// TwinCAT 3 PLC project Resi4MPM_Lib
// Title: Resi4MPM
// Company: Jan Wilch
// ProjectVersion: 1.0.0
// ProgramVersion: 3.1.4026.11
// libraries:
//   Tc2_Standard, * (Beckhoff Automation GmbH)
//   Tc2_System, * (Beckhoff Automation GmbH)
//   Tc3_Module, * (Beckhoff Automation GmbH)
// project tree:
//   Models/Behavior/ BehaviorBase.TcPOU, ControlPrimitiveBase.TcPOU, EBehaviorType.TcDUT, EOperationResult.TcDUT, ESpecialBehaviorIds.TcDUT, LinearSequence.TcPOU, ModuleSequenceBase.TcPOU
//   Models/Behavior/Strategy/ ESpecialStepIds.TcDUT, EStrategyStates.TcDUT, SStep.TcDUT, SStrategy.TcDUT, STransition.TcDUT
//   Models/ProcessState/AdsStateSynch/ SAdsSymbol.TcDUT
//   Models/ProcessState/ EDataType.TcDUT, HardwareObservationBase.TcPOU, ParameterSet.TcPOU, ProcessState.TcPOU, ProductBase.TcPOU, SNamedValue.TcDUT, SValue.TcDUT, UValues.TcDUT
//   Models/ProcessState/ProcessCondition/ BoolExpression.TcPOU, ComparisonExpression.TcPOU, EBoolOperation.TcDUT, EComparisonType.TcDUT, EExpressionType.TcDUT, IExpression.TcIO, IValExp.TcIO, SPrimitiveCondition.TcDUT, SBoolExpressionSpec.TcDUT, SInterlock.TcDUT, SConditionSpec.TcDUT, ValueExpression.TcPOU
//   Models/Reconfiguration/ EAbortState.TcDUT, ECompSeqState.TcDUT, ERecoveryState.TcDUT, ERetargetType.TcDUT, SCompensation.TcDUT, SRecovery.TcDUT, SRecoveryRequestOutput.TcDUT, SRetargeting.TcDUT, STriggeredOutput.TcDUT
//   / ResiConst.TcGVL
//   Services/Base/ ErrorManagerBase.TcPOU, ESeverity.TcDUT, ESpecialAlarmIds.TcDUT, IService.TcIO, SAlarm.TcDUT
//   Services/ ProcessManager.TcPOU, ServiceContainer.TcPOU, StateTracker.TcPOU
// real-time tasks:
//   TASK PlcTask: cycle T#10ms, priority 20, ADS port 350
//   TASK PlcTask1: cycle T#10ms, priority 23, ADS port 351
//   TASK PlcTask2: cycle T#10ms, priority 22, ADS port 352
//   TASK PlcTask3: cycle T#10ms, priority 21, ADS port 353

// ---- Models/Behavior/EBehaviorType.TcDUT
{attribute 'qualified_only'}
{attribute 'strict'}
TYPE EBehaviorType :
(
	none := 0,
	control_primitive := 1,
	user_sequence := 2,
	generated_sequence := 3
);
END_TYPE

// ---- Models/Behavior/EOperationResult.TcDUT
{attribute 'qualified_only'}
{attribute 'strict'}
TYPE EOperationResult :
(
	none := 0,
	success := 1,
	busy := 2,
	recovering := 3,
	waiting := 4,
	failed := 5,
	synced_success := 6
);
END_TYPE

// ---- Models/Behavior/ESpecialBehaviorIds.TcDUT
{attribute 'qualified_only'}
{attribute 'strict'}
TYPE ESpecialBehaviorIds :
(
	empty := 0,
	max_id := ResiConst.BEHAVIORS_ARR_MAX
) UINT;
END_TYPE

// ---- Models/Behavior/Strategy/ESpecialStepIds.TcDUT
{attribute 'qualified_only'}
{attribute 'strict'}
TYPE ESpecialStepIds :
(
	unset := -1,
	start := 0,
	end := 1
) INT;
END_TYPE

// ---- Models/Behavior/Strategy/EStrategyStates.TcDUT
{attribute 'qualified_only'}
{attribute 'strict'}
{attribute 'to_string'}
TYPE EStrategyStates :
(
	none := 0,
	ready := 1,
	running := 2,
	halting := 3,
	halted := 4,
	done := 5
) USINT;
END_TYPE

// ---- Models/Behavior/Strategy/SStep.TcDUT
{attribute 'OPC.UA.DA.StructuredType' := '1'}
TYPE SStep :
STRUCT
	// Set by the RA
	BehaviorType: EBehaviorType;
	BehaviorId: UINT;
	Parameters: ParameterSet;
	
	// defines ADS connections to step states on partner PLCs
	ExtSymbols: ARRAY [ResiConst.ARR_MIN..ResiConst.MAX_SYNC_PARTNERS] OF SAdsSymbol;
	// index of the responsible PLC (-1 is the current PLC is responsible)
	ExecutorIdx: INT;
	
	// Set by the PLC, read-only
	{attribute 'OPC.UA.DA.Access' := '1'}
	State: EOperationResult;
END_STRUCT
END_TYPE

// ---- Models/Behavior/Strategy/SStrategy.TcDUT
TYPE SStrategy :
STRUCT
	State: EStrategyStates;
	
	LoopStrategy: BOOL;
	Steps: ARRAY [ResiConst.ARR_MIN..ResiConst.STRAT_LEN_MAX] OF SStep;
	Transitions: ARRAY [ResiConst.ARR_MIN..ResiConst.STRAT_LEN_MAX] OF STransition;
	
	IsMaster: BOOL;
	NumPartners: UINT;
END_STRUCT
END_TYPE

// ---- Models/Behavior/Strategy/STransition.TcDUT
{attribute 'OPC.UA.DA.StructuredType' := '1'}
TYPE STransition :
STRUCT
	// determines whether this transition in a SStrategy's transition array is part of the strategy.
	IsSet: BOOL;
	
	// -1 signifies unset (because ID 0 is the start node)
	PrevStepIds: ARRAY [ResiConst.ARR_MIN..ResiConst.STRAT_PARALLEL_MAX] OF INT;
	// -1 signifies unset (because ID 0 is the start node)	
	NextStepIds: ARRAY [ResiConst.ARR_MIN..ResiConst.STRAT_PARALLEL_MAX] OF INT;
	
	ExpressionType: EExpressionType;
	ExpressionIdx: UINT;
END_STRUCT
END_TYPE

// ---- Models/ProcessState/AdsStateSynch/SAdsSymbol.TcDUT
TYPE SAdsSymbol :
STRUCT
	IsSet: BOOL;		// indicates whether this target is defined
	DataType: EDataType;
	
	NetId: T_AmsNetID;	// alias for STRING(23)
	Port: T_AmsPort;	// alias for UINT
	
	IdxGrp: UDINT;
	IdxOffs: UDINT;
END_STRUCT
END_TYPE

// ---- Models/ProcessState/EDataType.TcDUT
{attribute 'qualified_only'}
TYPE EDataType :
(
	none := 0,
	dont_care := 1,
	binary := 2,
	numeric := 3,
	string_t := 4
) USINT;
END_TYPE

// ---- Models/ProcessState/ProcessCondition/EBoolOperation.TcDUT
{attribute 'qualified_only'}
{attribute 'strict'}
TYPE EBoolOperation :
(
	none := 0,
	and_op := 1,
	nand_op := 2,
	or_op := 3,
	nor_op := 4
);
END_TYPE

// ---- Models/ProcessState/ProcessCondition/EComparisonType.TcDUT
{attribute 'qualified_only'}
{attribute 'strict'}
TYPE EComparisonType :
(
	none := 0,
	equals := 1,
	not_equal := 2,
	greater := 3,
	less := 4,
	greater_eq := 5,
	less_eq := 6
);
END_TYPE

// ---- Models/ProcessState/ProcessCondition/EExpressionType.TcDUT
{attribute 'qualified_only'}
{attribute 'strict'}
TYPE EExpressionType :
(
	none := 0,
	boolean := 1,
	comparison := 2,
	value := 3
);
END_TYPE

// ---- Models/ProcessState/ProcessCondition/SPrimitiveCondition.TcDUT
TYPE SPrimitiveCondition EXTENDS SConditionSpec :
STRUCT
	PrimitiveId: UINT;
	// if it's not a precondition, it's a postcondition
	IsPre: BOOL;
END_STRUCT
END_TYPE

// ---- Models/ProcessState/ProcessCondition/SBoolExpressionSpec.TcDUT
{attribute 'OPC.UA.DA.StructuredType' := '1'}
TYPE SBoolExpressionSpec :
STRUCT
	Operator: EBoolOperation;
	
	LeftType: EExpressionType;
	LeftIdx: UINT;
	
	RightType: EExpressionType;
	RightIdx: UINT;
END_STRUCT
END_TYPE

// ---- Models/ProcessState/ProcessCondition/SInterlock.TcDUT
TYPE SInterlock EXTENDS SConditionSpec :
STRUCT
	DefaultValue: BOOL;
END_STRUCT
END_TYPE

// ---- Models/ProcessState/ProcessCondition/SConditionSpec.TcDUT
{attribute 'OPC.UA.DA.StructuredType' := '1'}
TYPE SConditionSpec :
STRUCT
	IsActive: BOOL;
	ExpressionType: EExpressionType;
	ExpressionIdx: UINT;
END_STRUCT
END_TYPE

// ---- Models/ProcessState/SNamedValue.TcDUT
{attribute 'OPC.UA.DA.StructuredType' := '1'}
TYPE SNamedValue EXTENDS SValue :
STRUCT
	Name: STRING;
END_STRUCT
END_TYPE

// ---- Models/ProcessState/SValue.TcDUT
TYPE SValue :
STRUCT
	DataType: EDataType;
	Value: UValues;
	Defined: BOOL;
END_STRUCT
END_TYPE

// ---- Models/ProcessState/UValues.TcDUT
TYPE UValues :
UNION
	Binary: BOOL;
	Numeric: LREAL;
	String_t: STRING;
END_UNION
END_TYPE

// ---- Models/Reconfiguration/EAbortState.TcDUT
{attribute 'qualified_only'}
{attribute 'strict'}
TYPE EAbortState :
(
	none := 0,
	requested := 1,
	aborting := 2,
	aborted := 3
);
END_TYPE

// ---- Models/Reconfiguration/ECompSeqState.TcDUT
{attribute 'qualified_only'}
{attribute 'strict'}
TYPE ECompSeqState :
(
	none := 0,
	preparing := 1,
	running := 2,
	finished := 3
);
END_TYPE

// ---- Models/Reconfiguration/ERecoveryState.TcDUT
{attribute 'qualified_only'}
{attribute 'strict'}
TYPE ERecoveryState :
(
	none := 0,
	requested := 1,
	awaiting := 2,
	running := 3,
	completed := 4,
	failed := 5
);
END_TYPE

// ---- Models/Reconfiguration/ERetargetType.TcDUT
{attribute 'qualified_only'}
{attribute 'strict'}
TYPE ERetargetType :
(
	not_retargeted := 0,
	primitive_target := 1,
	sequence_target := 2
);
END_TYPE

// ---- Models/Reconfiguration/SCompensation.TcDUT
{attribute 'OPC.UA.DA.StructuredType' := '1'}
TYPE SCompensation :
STRUCT
	IsActive: BOOL;	

	(* ID of the Control Primitive that cannot operate anymore. *)
	SickPrimitiveId: UINT;
	
	(* Specifies whether the sick primitive is replaced by another primitive or a sequence. *)
	NewType: EBehaviorType;
	
	(* If NewType is primitive or user-sequence: ID of the sick primitive's replacement. *)
	NewId: UINT;
	
	(* If needed, parameters that are set (or overwritten) before executing the replacement.
	   For replacement types primtive or user-generated sequence, only the first element is used. *)
	ParameterSets: ARRAY [ResiConst.ARR_MIN..ResiConst.MODULE_SEQ_ARR_MAX] OF ParameterSet;
	
	(* If NewType is generated sequence: The (linear) sequence of copmensation primitives. *)
	PrimitiveIds: ARRAY [ResiConst.ARR_MIN..ResiConst.MODULE_SEQ_ARR_MAX] OF UINT;
END_STRUCT
END_TYPE

// ---- Models/Reconfiguration/SRecovery.TcDUT
{attribute 'OPC.UA.DA.StructuredType' := '1'}
TYPE SRecovery :
STRUCT
	(* The sequence of Control Primitives to execute for recovery or defining.*)
	RecoveryStrategy: ARRAY [ResiConst.ARR_MIN..ResiConst.MODULE_SEQ_ARR_MAX] OF UINT;
	
	(* The parameters needed by the strategy's primitives. *)
	RecoveryParameters: ParameterSet;
END_STRUCT
END_TYPE

// ---- Models/Reconfiguration/SRecoveryRequestOutput.TcDUT
{attribute 'OPC.UA.DA.StructuredType' := '1'}
TYPE SRecoveryRequestOutput EXTENDS STriggeredOutput :
STRUCT
	RequestedState: STRING(256);
END_STRUCT
END_TYPE

// ---- Models/Reconfiguration/SRetargeting.TcDUT
TYPE SRetargeting :
STRUCT
	RetargetType: ERetargetType;
	TargetId: UINT;
	// parameters that are set or overwritten before the primitive is executed
	OverwriteParams: ParameterSet;
END_STRUCT
END_TYPE

// ---- Models/Reconfiguration/STriggeredOutput.TcDUT
TYPE STriggeredOutput :
STRUCT
	ChangeTrigger: USINT;
END_STRUCT
END_TYPE

// ---- Services/Base/ESeverity.TcDUT
{attribute 'qualified_only'}
{attribute 'strict'}
TYPE ESeverity :
(
	none := 0,
	info := 1,
	warning := 2,
	error := 3
) UINT;
END_TYPE

// ---- Services/Base/ESpecialAlarmIds.TcDUT
{attribute 'qualified_only'}
{attribute 'strict'}
TYPE ESpecialAlarmIds :
(
	none := 0,
	recovery_request := 990,
	definition_request := 991,
	strategy_received := 992
) UINT;
END_TYPE

// ---- Services/Base/SAlarm.TcDUT
(*
 * see: https://www.plcnext.help/te/Service_Components/Alarms/Alarms_via_OPC_UA.htm
 *)
{attribute 'OPC.UA.DA.StructuredType' := '1'}
TYPE SAlarm :
STRUCT
	// Time in number of 100 ns intervals since 01.01.1601.
	TimeTicks: ULINT;
	AlarmId: UINT;
	// TODO - AlarmType
	Active: BOOL;
	//Acknowledged: BOOL;
	//Confirmed: BOOL;
	Severity: ESeverity;
	//RetainAlarm: BOOL;
	Message: STRING;
	InstanceName: STRING;
END_STRUCT
END_TYPE

// ---- ResiConst.TcGVL
{attribute 'qualified_only'}
VAR_GLOBAL CONSTANT	
	// Lower bound of all Resi4MPM arrays.
	ARR_MIN: UINT := 0;
	// Default upper bound of Resi4MPM arrays.
	DEFAULT_ARR_MAX: UINT := 10;
	// Max length of behaviors (separately length of Control Primitives and Module Sequences).
	BEHAVIORS_ARR_MAX: UINT := 100;
	// Max length of observed process variables.
	STATE_ARR_MAX: UINT := 150;
	// Max length of units observing the process state.
	OBSERVERS_ARR_MAX: UINT := 100;
	// Max length of UC-C strategies introduced at runtime.
	COMPENSATIONS_ARR_MAX: UINT := 10;
	// Max Control Primitive count of Module Sequences.
	MODULE_SEQ_ARR_MAX: UINT := 10;
	// Max number of parameters for a Behavior.
	PARAMS_ARR_MAX: UINT := 10;
	// Max number of Products 
	PRODUCTS_ARR_MAX: UINT := 20;
	// Max number of parallel steps in a runtime-defined strategy.
	STRAT_PARALLEL_MAX: UINT := 5;
	// Max length (number of steps/transitions) of a runtime-defined strategy.
	STRAT_LEN_MAX: UINT := 24;
	// Max length of runtime-changeable expressions.
	RT_EXPRS_MAX: UINT := 24;
	// Maximum number of synchronized foreign PLCs.
	MAX_SYNC_PARTNERS: UINT := 5;
END_VAR

// ---- Models/ProcessState/ProcessCondition/IExpression.TcIO
INTERFACE IExpression EXTENDS __System.IQueryInterface

METHOD IsTrue : BOOL
VAR_INPUT
	i_ptrProcessState: POINTER TO ProcessState;
END_VAR
END_METHOD

METHOD ToString : STRING(256)
VAR_INPUT
END_VAR
END_METHOD

END_INTERFACE

// ---- Models/ProcessState/ProcessCondition/IValExp.TcIO
// this interface is only necessary to allow type-checking for Value Expressions
INTERFACE IValExp EXTENDS __System.IQueryInterface

END_INTERFACE

// ---- Services/Base/IService.TcIO
INTERFACE IService

END_INTERFACE

// ---- Models/Behavior/BehaviorBase.TcPOU
(* Common base of all reusable behavior types. *)
FUNCTION_BLOCK ABSTRACT BehaviorBase
VAR_INPUT
	i_params: ParameterSet;
END_VAR
VAR_OUTPUT
	{attribute 'OPC.UA.DA' := '1'}
	{attribute 'OPC.UA.DA.Access' := '1'}
	o_status: EOperationResult;
END_VAR
VAR
	(* Because all Control Primitives and Module Sequences instances are 
       singletons, they can set their IDs themselves *)
	{attribute 'OPC.UA.DA' := '1'}
	{attribute 'OPC.UA.DA.Access' := '1'}
	m_id: UINT;
	
	(* define's the behavior's parameters (if any)
	   format: <Name1>:<Type1>;<Name2>:<Type2>;... *)
	{attribute 'OPC.UA.DA' := '1'}
	{attribute 'OPC.UA.DA.Access' := '1'}
	m_paramDefinition: STRING;
END_VAR

PROPERTY Id : UINT
GET
Id := m_id;
END_GET
END_PROPERTY

PROPERTY ABSTRACT Postcondition : IExpression
GET
END_GET
END_PROPERTY

PROPERTY ABSTRACT Precondition : IExpression
GET
END_GET
END_PROPERTY

END_FUNCTION_BLOCK

// ---- Models/ProcessState/ParameterSet.TcPOU
FUNCTION_BLOCK ParameterSet
VAR_INPUT
END_VAR
VAR_OUTPUT
END_VAR
VAR
	m_parameters : ARRAY [ResiConst.ARR_MIN..ResiConst.PARAMS_ARR_MAX] OF SNamedValue;
END_VAR

PROPERTY Parameters : ARRAY [ResiConst.ARR_MIN..ResiConst.PARAMS_ARR_MAX] OF SNamedValue
GET
Parameters := m_parameters;
END_GET
END_PROPERTY

METHOD Reset : BOOL
VAR
	emptyVal: UValues;
	i: UINT;
END_VAR
FOR i := ResiConst.ARR_MIN TO ResiConst.PARAMS_ARR_MAX DO
	m_parameters[i].DataType := EDataType.none;
	m_parameters[i].Defined := FALSE;
	m_parameters[i].Name := '';
	m_parameters[i].Value := emptyVal;
END_FOR
END_METHOD

METHOD Retrieve : SNamedValue
VAR_INPUT
	i_name: STRING;
END_VAR
VAR
	i: UINT;
	m_emptyParam: SNamedValue;
END_VAR
FOR i := ResiConst.ARR_MIN TO ResiConst.PARAMS_ARR_MAX DO
	IF m_parameters[i].Name = i_name THEN
		Retrieve := m_parameters[i];
		RETURN;
	END_IF
END_FOR

Retrieve := m_emptyParam;
END_METHOD

METHOD SetParam_Binary : BOOL
VAR_INPUT
	i_key: STRING;
	i_value: BOOL;
END_VAR
VAR
	i: UINT;
	m_paramFound: BOOL;
	nonEmptyIdx: UINT;
END_VAR
FOR i := 0 TO ResiConst.PARAMS_ARR_MAX DO
	IF m_parameters[i].Name = i_key THEN
		m_parameters[i].DataType := EDataType.binary;
		m_parameters[i].Value.Binary := i_value;
		m_paramFound := TRUE;
	ELSIF m_parameters[i].Name <> '' THEN
		nonEmptyIdx := i;
	ELSE
		EXIT;
	END_IF
END_FOR

IF NOT m_paramFound THEN
	m_parameters[nonEmptyIdx + 1].DataType := EDataType.binary;
	m_parameters[nonEmptyIdx + 1].Value.Binary := i_value;
	m_parameters[nonEmptyIdx + 1].Name := i_key;
END_IF
END_METHOD

METHOD SetParam_Defined : BOOL
VAR_INPUT
	i_key: STRING;
	i_defined: BOOL;
END_VAR
VAR
	i: UINT;
	m_paramsFound: BOOL;	
END_VAR
FOR i := 0 TO ResiConst.PARAMS_ARR_MAX DO
	IF m_parameters[i].Name = i_key THEN
		m_parameters[i].Defined := i_defined;
		m_paramsFound := TRUE;
		SetParam_Defined := TRUE;
	END_IF
END_FOR

IF NOT m_paramsFound THEN
	SetParam_Defined := FALSE;
END_IF
END_METHOD

METHOD SetParam_Numeric : BOOL
VAR_INPUT
	i_key: STRING;
	i_value: LREAL;
END_VAR
VAR
	i: UINT;
	m_paramFound: BOOL;
	nonEmptyIdx: UINT;
END_VAR
FOR i := 0 TO ResiConst.PARAMS_ARR_MAX DO
	IF m_parameters[i].Name = i_key THEN
		m_parameters[i].DataType := EDataType.numeric;
		m_parameters[i].Value.Numeric := i_value;
		m_paramFound := TRUE;
	ELSIF m_parameters[i].Name <> '' THEN
		nonEmptyIdx := i;
	ELSE
		EXIT;
	END_IF
END_FOR

IF NOT m_paramFound THEN
	m_parameters[nonEmptyIdx + 1].DataType := EDataType.numeric;
	m_parameters[nonEmptyIdx + 1].Value.Numeric := i_value;
	m_parameters[nonEmptyIdx + 1].Name := i_key;
END_IF
END_METHOD

METHOD SetParam_String : BOOL
VAR_INPUT
	i_key: STRING;
	i_value: STRING;
END_VAR
VAR
	i: UINT;
	m_paramFound: BOOL;
	nonEmptyIdx: UINT;
END_VAR
FOR i := 0 TO ResiConst.PARAMS_ARR_MAX DO
	IF m_parameters[i].Name = i_key THEN
		m_parameters[i].DataType := EDataType.string_t;
		m_parameters[i].Value.String_t := i_value;
		m_paramFound := TRUE;
	ELSIF m_parameters[i].Name <> '' THEN
		nonEmptyIdx := i;
	ELSE
		EXIT;
	END_IF
END_FOR

IF NOT m_paramFound THEN
	m_parameters[nonEmptyIdx + 1].DataType := EDataType.string_t;
	m_parameters[nonEmptyIdx + 1].Value.String_t := i_value;
	m_parameters[nonEmptyIdx + 1].Name := i_key;
END_IF
END_METHOD

END_FUNCTION_BLOCK

// ---- Models/Behavior/ControlPrimitiveBase.TcPOU
(* Base of Control Primitives. Inheriting FBs must implement the type-specific "ExecuteInternal" method. *)
FUNCTION_BLOCK ABSTRACT ControlPrimitiveBase EXTENDS BehaviorBase
VAR
	m_timeout: TIME;
	
	m_internalRes: BOOL;
	m_pre: IExpression;
	m_post: IExpression;
	
	// store the conditions as string for access via OPC UA + easier debugging
	{attribute 'OPC.UA.DA' := '1'}
	{attribute 'OPC.UA.DA.Access' := '1'}
	m_preStr: STRING(256);
	{attribute 'OPC.UA.DA' := '1'}
	{attribute 'OPC.UA.DA.Access' := '1'}
	m_postStr: STRING(256);
	
	m_st: POINTER TO StateTracker;
	m_pm: POINTER TO ProcessManager;
	
	m_tonTimeout: TON;
	
	m_didAbort: BOOL;
END_VAR

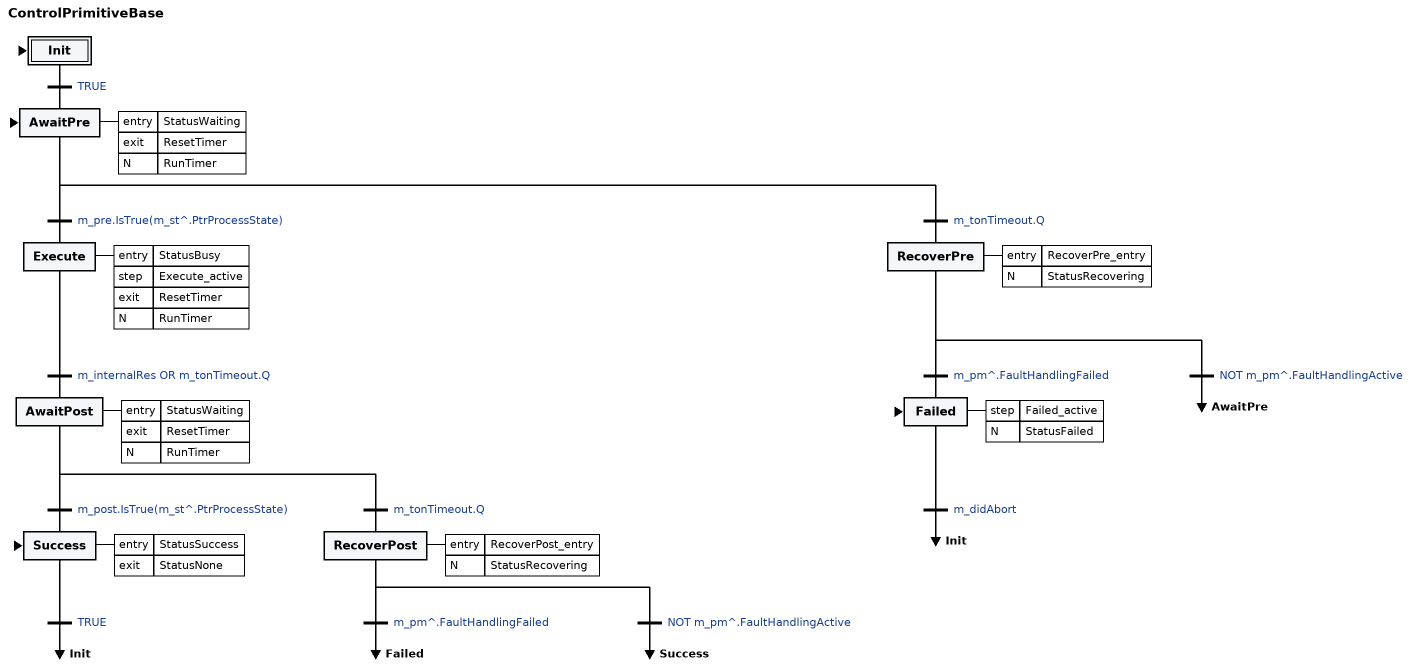
INITIAL_STEP Init:
END_STEP
TRANSITION FROM Init TO AwaitPre
    := TRUE;
END_TRANSITION
STEP AwaitPre:
    StatusWaiting(P1);  // entry action
    ResetTimer(P0);  // exit action
    RunTimer(N);
END_STEP
TRANSITION FROM AwaitPre TO Execute
    := m_pre.IsTrue(m_st^.PtrProcessState);
END_TRANSITION
STEP Execute:
    StatusBusy(P1);  // entry action
    Execute_active(N);  // step action
    ResetTimer(P0);  // exit action
    RunTimer(N);
END_STEP
TRANSITION FROM Execute TO AwaitPost
    := m_internalRes OR m_tonTimeout.Q;
END_TRANSITION
STEP AwaitPost:
    StatusWaiting(P1);  // entry action
    ResetTimer(P0);  // exit action
    RunTimer(N);
END_STEP
TRANSITION FROM AwaitPost TO Success
    := m_post.IsTrue(m_st^.PtrProcessState);
END_TRANSITION
STEP Success:
    StatusSuccess(P1);  // entry action
    StatusNone(P0);  // exit action
END_STEP
TRANSITION FROM Success TO Init
    := TRUE;
END_TRANSITION
TRANSITION FROM AwaitPost TO RecoverPost
    := m_tonTimeout.Q;
END_TRANSITION
STEP RecoverPost:
    RecoverPost_entry(P1);  // entry action
    StatusRecovering(N);
END_STEP
TRANSITION FROM RecoverPost TO Failed
    := m_pm^.FaultHandlingFailed;
END_TRANSITION
TRANSITION FROM RecoverPost TO Success
    := NOT m_pm^.FaultHandlingActive;
END_TRANSITION
TRANSITION FROM AwaitPre TO RecoverPre
    := m_tonTimeout.Q;
END_TRANSITION
STEP RecoverPre:
    RecoverPre_entry(P1);  // entry action
    StatusRecovering(N);
END_STEP
TRANSITION FROM RecoverPre TO Failed
    := m_pm^.FaultHandlingFailed;
END_TRANSITION
STEP Failed:
    Failed_active(N);  // step action
    StatusFailed(N);
END_STEP
TRANSITION FROM Failed TO Init
    := m_didAbort;
END_TRANSITION
TRANSITION FROM RecoverPre TO AwaitPre
    := NOT m_pm^.FaultHandlingActive;
END_TRANSITION

METHOD ABSTRACT Abort : BOOL
VAR_INPUT
END_VAR
END_METHOD

ACTION Execute_active:
IF NOT m_internalRes THEN
	m_internalRes := ExecuteInternal(i_params);
END_IF
END_ACTION

(* Execution logic of this Control Primitive. *)
METHOD PROTECTED ABSTRACT ExecuteInternal : BOOL
VAR_INPUT
	i_params: ParameterSet;
END_VAR
END_METHOD

ACTION Failed_active:
m_didAbort := Abort();
END_ACTION

PROPERTY Postcondition : IExpression
GET
Postcondition := m_post;
END_GET
SET
m_post := Postcondition;
m_postStr := Postcondition.ToString();
END_SET
END_PROPERTY

PROPERTY Precondition : IExpression
GET
Precondition := m_pre;
END_GET
SET
m_pre := Precondition;
m_preStr := Precondition.ToString();
END_SET
END_PROPERTY

METHOD ProvideServices : BOOL
VAR_INPUT
	i_ptrProcessManager: POINTER TO ProcessManager;
	i_ptrStateTracker: POINTER TO StateTracker;
END_VAR
m_pm := i_ptrProcessManager;
m_st := i_ptrStateTracker;
END_METHOD

ACTION RecoverPost_entry:
m_pm^.RequestRecovery(m_post, CONCAT('Primitive ', TO_STRING(m_id)));
END_ACTION

ACTION RecoverPre_entry:
m_pm^.RequestRecovery(m_pre, CONCAT('Primitive ', TO_STRING(m_id)));
END_ACTION

ACTION ResetTimer:
m_tonTimeout(IN := FALSE);
m_internalRes := FALSE;
END_ACTION

ACTION RunTimer:
m_tonTimeout(IN := TRUE, PT := m_timeout);
END_ACTION

ACTION StatusBusy:
o_status := EOperationResult.busy;
END_ACTION

ACTION StatusFailed:
o_status := EOperationResult.failed;
END_ACTION

ACTION StatusNone:
o_status := EOperationResult.none;
END_ACTION

ACTION StatusRecovering:
o_status := EOperationResult.recovering;
END_ACTION

ACTION StatusSuccess:
o_status := EOperationResult.success;
END_ACTION

ACTION StatusWaiting:
o_status := EOperationResult.waiting;
END_ACTION

END_FUNCTION_BLOCK

// ---- Services/StateTracker.TcPOU
FUNCTION_BLOCK StateTracker IMPLEMENTS IService
VAR
	// ***** OUTPUT TO RA (read-only) ******
	{attribute 'OPC.UA.DA' := '1'}
	{attribute 'OPC.UA.DA.Access' := '1'}
	// locally monitored variables AND non-local variables synced via ADS
	raInOut_processState: ARRAY [ResiConst.ARR_MIN..ResiConst.STATE_ARR_MAX] OF SNamedValue;
	
	{attribute 'OPC.UA.DA' := '1'}
	raIn_stateSyncTargets: 	ARRAY [ResiConst.ARR_MIN..ResiConst.STATE_ARR_MAX] OF SAdsSymbol;
	// *************************
	
	m_ptrProcessManager: POINTER TO ProcessManager;
	m_completeState: ProcessState;
	
	// POUs capable of observing part of the process state
	m_hwObsIdx: UINT := 0;
	m_hwObservations: ARRAY [ResiConst.ARR_MIN..ResiConst.OBSERVERS_ARR_MAX] OF POINTER TO HardwareObservationBase;
	
	(*  PRODUCT MANAGEMENT
		Manages the flow of (discrete) products through the process by shifting product information between array places. *)
	m_productBases: ARRAY [ResiConst.ARR_MIN..ResiConst.PRODUCTS_ARR_MAX] OF ProductBase;
	m_productPtrs: ARRAY [ResiConst.ARR_MIN..ResiConst.PRODUCTS_ARR_MAX] OF POINTER TO ProductBase;
	
	// INTERLOCKS
	m_interlocks: ARRAY [ResiConst.ARR_MIN..ResiConst.COMPENSATIONS_ARR_MAX] OF IExpression;
	m_interlockIdx: UINT;
	m_expectedVals: ARRAY [ResiConst.ARR_MIN..ResiConst.COMPENSATIONS_ARR_MAX] OF BOOL;
	
	// ADS SYNCH
	m_stateReaders: ARRAY [ResiConst.ARR_MIN..ResiConst.STATE_ARR_MAX] OF ADSREAD;
END_VAR

METHOD AddInterlock : BOOL
VAR_INPUT
	i_interlock: IExpression;
	i_expectedVal: BOOL;
END_VAR
m_interlocks[m_interlockIdx] := i_interlock;
m_expectedVals[m_interlockIdx] := i_expectedVal;
m_interlockIdx := m_interlockIdx + 1;
END_METHOD

METHOD AddObservation : BOOL
VAR_INPUT
	i_ptrObservation: POINTER TO HardwareObservationBase;
END_VAR
m_hwObservations[m_hwObsIdx] := i_ptrObservation;
m_hwObsIdx := m_hwObsIdx + 1;
END_METHOD

METHOD CyclicUpdateStatus : BOOL
VAR_INPUT
	i_ignoreDefinition: BOOL;
END_VAR
VAR_IN_OUT
	// Variables that are observable only at app-level. 
	// NOTE: The index is interpreted as the process variable ID.
	io_appLevelVars: ARRAY[*] OF SValue;
END_VAR
VAR
	ui: UINT;
	di: DINT;
	m_tmpVal: SValue;
	m_otherVal: SValue;
	m_sym: SAdsSymbol;
	m_len: UDINT;
	m_adr: PVOID;
END_VAR
// apply the process-level observation (e.g., current operation mode or recipe step)
FOR di := LOWER_BOUND(io_appLevelVars, 1) TO UPPER_BOUND(io_appLevelVars, 1) DO
	m_completeState.SetValue(DINT_TO_UINT(di), io_appLevelVars[di]);
END_FOR

// update hardware-level observation
FOR ui := ResiConst.ARR_MIN TO ResiConst.OBSERVERS_ARR_MAX DO
	IF m_hwObservations[ui] <> 0 THEN
		m_hwObservations[ui]^.UpdateProcessObservation(THIS^.m_completeState);
	END_IF
END_FOR

FOR ui := ResiConst.ARR_MIN TO (ResiConst.DEFAULT_ARR_MAX)DO
	m_productPtrs[ui]^.UpdateProcessObservation(THIS^.m_completeState);
END_FOR

IF i_ignoreDefinition THEN
	FOR ui := ResiConst.ARR_MIN TO ResiConst.STATE_ARR_MAX DO
		m_completeState.UpdateState_Defined(ui, TRUE);
	END_FOR
END_IF

// check interlocks
FOR ui := ResiConst.ARR_MIN TO ResiConst.COMPENSATIONS_ARR_MAX DO
	IF m_interlocks[ui] <> 0 THEN
		IF m_interlocks[ui].IsTrue(ADR(m_completeState)) <> m_expectedVals[ui] AND NOT m_ptrProcessManager^.AbortActive THEN
			// interlock violated -> abort all
			m_ptrProcessManager^.RequestAbort();
			RETURN;
		END_IF
	END_IF
END_FOR

// synch with other PLCs
FOR ui := ResiConst.ARR_MIN TO ResiConst.STATE_ARR_MAX DO
	m_sym := raIn_stateSyncTargets[ui];
	IF m_sym.IsSet THEN
		// use the raInOut_processState as a buffer; copy to the actual process state (at least one cycle delayed)
		m_tmpVal.DataType := m_sym.DataType;
		m_tmpVal.Defined := TRUE;	// TODO (?) - copy the actual Defined flags
		CASE m_sym.DataType OF
			EDataType.binary:
				m_len := SIZEOF(raInOut_processState[ui].Value.Binary);
				m_adr := ADR(raInOut_processState[ui].Value.Binary);
				m_tmpVal.Value.Binary := raInOut_processState[ui].Value.Binary;
			EDataType.numeric:
				m_len := SIZEOF(raInOut_processState[ui].Value.Numeric);
				m_adr := ADR(raInOut_processState[ui].Value.Numeric);
				m_tmpVal.Value.Numeric := raInOut_processState[ui].Value.Numeric;
			EDataType.string_t:
				m_len := SIZEOF(raInOut_processState[ui].Value.String_t);
				m_adr := ADR(raInOut_processState[ui].Value.String_t);
				m_tmpVal.Value.String_t := raInOut_processState[ui].Value.String_t;
		END_CASE
		
		m_stateReaders[ui](READ := FALSE);
		m_stateReaders[ui](
			NETID := raIn_stateSyncTargets[ui].NetId,
			PORT := raIn_stateSyncTargets[ui].Port,
			IDXGRP := m_sym.IdxGrp,
			IDXOFFS := m_sym.IdxOffs,
			LEN := m_len,
			DESTADDR := m_adr,
			READ := TRUE);
			
		m_completeState.SetValue(ui, m_tmpVal);
	END_IF
END_FOR

// RA output
FOR ui := ResiConst.ARR_MIN TO ResiConst.STATE_ARR_MAX DO
	m_tmpVal := m_completeState.Retrieve(ui, FALSE);
	raInOut_processState[ui].DataType := m_tmpVal.DataType;
	raInOut_processState[ui].Value.Binary := m_tmpVal.Value.Binary;
	raInOut_processState[ui].Value.Numeric := m_tmpVal.Value.Numeric;
	raInOut_processState[ui].Value.String_t := m_tmpVal.Value.String_t;
	raInOut_processState[ui].Defined := m_tmpVal.Defined;
END_FOR
END_METHOD

//FB_Init is always available implicitly and it is used primarily for initialization.
//The return value is not evaluated. For a specific influence, you can also declare the
//methods explicitly and provide additional code there with the standard initialization
//code. You can evaluate the return value.
METHOD FB_Init: BOOL
VAR_INPUT
    bInitRetains: BOOL; // TRUE: the retain variables are initialized (reset warm / reset cold)
    bInCopyCode: BOOL;  // TRUE: the instance will be copied to the copy code afterward (online change)   
END_VAR
VAR
	i: UINT;
END_VAR
FOR i := ResiConst.ARR_MIN TO ResiConst.DEFAULT_ARR_MAX DO
	m_productPtrs[i] := ADR(m_productBases[i]);
END_FOR
END_METHOD

METHOD GetBinary : BOOL
VAR_INPUT
	i_processVariableId: UINT;
END_VAR
VAR
	m_value: SValue;
END_VAR
m_value := m_completeState.Retrieve(i_processVariableId, TRUE);
GetBinary := m_value.Value.Binary;
END_METHOD

METHOD GetDefined : BOOL
VAR_INPUT
	i_processVariableId: UINT;
END_VAR
VAR
	m_value: SValue;
END_VAR
m_value := m_completeState.Retrieve(i_processVariableId, FALSE);
GetDefined := m_value.Defined;
END_METHOD

METHOD GetNumeric : LREAL
VAR_INPUT
	i_processVariableId: UINT;
END_VAR
VAR
	m_value: SValue;
END_VAR
m_value := m_completeState.Retrieve(i_processVariableId, TRUE);
GetNumeric := m_value.Value.Numeric;
END_METHOD

METHOD GetString : STRING
VAR_INPUT
	i_processVariableId: UINT;
END_VAR
VAR
	m_value: SValue;
END_VAR
m_value := m_completeState.Retrieve(i_processVariableId, TRUE);
GetString := m_value.Value.String_t;
END_METHOD

METHOD ProvideServices : BOOL
VAR_INPUT
	i_ptrProcessManager: POINTER TO ProcessManager;
END_VAR
THIS^.m_ptrProcessManager := i_ptrProcessManager;
m_completeState.ProvideServices(i_ptrProcessManager);
END_METHOD

PROPERTY PtrProcessState : POINTER TO ProcessState
GET
PtrProcessState := ADR(m_completeState);
END_GET
END_PROPERTY

METHOD RegisterLocalProduct : BOOL
VAR_INPUT
	i_productID: UINT;
	i_productPtr: POINTER TO ProductBase;
END_VAR
m_productPtrs[i_productID] := i_productPtr;

// copy the
END_METHOD

METHOD ResetConfiguration : BOOL
VAR
	i: UINT;
	emptySym: SAdsSymbol;
	emptyExpr: IExpression;
END_VAR
FOR i := ResiConst.ARR_MIN TO ResiConst.STATE_ARR_MAX DO
	raIn_stateSyncTargets[i] := emptySym;
END_FOR

FOR i := ResiConst.ARR_MIN TO ResiConst.PRODUCTS_ARR_MAX DO
	m_productBases[i].ResetConfiguration();
END_FOR

m_interlockIdx := 0;
FOR i := ResiConst.ARR_MIN TO ResiConst.COMPENSATIONS_ARR_MAX DO
	m_interlocks[i] := emptyExpr;
	m_expectedVals[i] := FALSE;
END_FOR
END_METHOD

METHOD ResetDefinitions : BOOL
VAR_INPUT
END_VAR
VAR 
	i: UINT;
END_VAR
FOR i := ResiConst.ARR_MIN TO ResiConst.OBSERVERS_ARR_MAX DO
	IF m_hwObservations[i] <> 0 THEN
		m_hwObservations[i]^.ResetDefinition();
	END_IF
END_FOR
END_METHOD

METHOD SetProcessVariableName : BOOL
VAR_INPUT
	var_idx: UINT;
	name: STRING;
END_VAR
raInOut_processState[var_idx].Name := name;
END_METHOD

METHOD ShiftProduct : BOOL
VAR_INPUT
	i_srcID: UINT;
	i_dstID: UINT;
END_VAR
ShiftProduct := FALSE;

IF m_productPtrs[i_dstID]^.Copy(m_productPtrs[i_srcID]) THEN
	m_productPtrs[i_srcID]^.Reset();
	ShiftProduct := TRUE;
END_IF
END_METHOD

END_FUNCTION_BLOCK

// ---- Services/ProcessManager.TcPOU
FUNCTION_BLOCK ProcessManager IMPLEMENTS IService
VAR_INPUT
END_VAR
VAR_OUTPUT
END_VAR
VAR
	// ***** INPUT FROM RA *****
	{attribute 'OPC.UA.DA' := '1'}
	raIn_compensations: ARRAY [ResiConst.ARR_MIN..ResiConst.COMPENSATIONS_ARR_MAX] OF SCompensation;
	
	{attribute 'OPC.UA.DA' := '1'}
	raIn_recoveryAvailable: BOOL;
	{attribute 'OPC.UA.DA' := '1'}
	raIn_recovery: SRecovery;
	
	{attribute 'OPC.UA.DA' := '1'}
	raIn_valueExpressions: ARRAY [ResiConst.ARR_MIN..ResiConst.RT_EXPRS_MAX] OF ValueExpression(EDataType.none, FALSE, 0, '', FALSE);
	{attribute 'OPC.UA.DA' := '1'}
	raIn_compExpressions: ARRAY [ResiConst.ARR_MIN..ResiConst.RT_EXPRS_MAX] OF ComparisonExpression(0, EComparisonType.none, EDataType.none, FALSE, 0, '', FALSE);
	{attribute 'OPC.UA.DA' := '1'}
	raIn_boolExprSpecs: ARRAY [ResiConst.ARR_MIN..ResiConst.RT_EXPRS_MAX] OF SBoolExpressionSpec;
	
	{attribute 'OPC.UA.DA' := '1'}
	raIn_runtimeConditions: ARRAY [ResiConst.ARR_MIN..ResiConst.COMPENSATIONS_ARR_MAX] OF SPrimitiveCondition;
	{attribute 'OPC.UA.DA' := '1'}
	raIn_runtimeInterlocks: ARRAY [ResiConst.ARR_MIN..ResiConst.COMPENSATIONS_ARR_MAX] OF SInterlock;
	
	{attribute 'OPC.UA.DA' := '1'}
	raIn_customStrategy: SStrategy;	
	// *************************
	
	// ***** OUTPUT TO RA (read-only) ******
	{attribute 'OPC.UA.DA' := '1'}
	{attribute 'OPC.UA.DA.Access' := '1'}
	raOut_recoveryRequest: SRecoveryRequestOutput;
	// *************************
	
	m_ptrStateTracker: POINTER TO StateTracker;
	m_ptrErrorMgr: POINTER TO ErrorManagerBase;
	
	m_trueValue: ValueExpression(EDataType.binary, TRUE, 0, '', TRUE);
	m_ptrPrimitives: ARRAY [ResiConst.ARR_MIN..ResiConst.BEHAVIORS_ARR_MAX] OF POINTER TO ControlPrimitiveBase;
	
	(* Half of the array is reserved for user-defined sequences, the other for runtime-defined compensations. *)
	m_ptrSequences: ARRAY [ResiConst.ARR_MIN..2 * ResiConst.BEHAVIORS_ARR_MAX] OF POINTER TO ModuleSequenceBase;
	
	(* COMPENSATION
	   Array index: ID of the sick Control Primitive.
	   Array entry: specification of the primitive/sequence that should be executed instead. *)
	m_retargets: ARRAY [ResiConst.ARR_MIN..ResiConst.BEHAVIORS_ARR_MAX] OF SRetargeting;
	
	// compensation sequences that can be defined at runtime
	m_compSeqs: ARRAY [ResiConst.BEHAVIORS_ARR_MAX + 1..ResiConst.BEHAVIORS_ARR_MAX + ResiConst.COMPENSATIONS_ARR_MAX] OF LinearSequence;
	m_compSeqsIdx: UINT := ResiConst.BEHAVIORS_ARR_MAX + 1;
	m_activeCompensationState: ECompSeqState;
	m_activeCompensationIdx: UINT;
	
	(* RECOVERY / DEFINITION *)
	m_conditionToRecover: IExpression;
	m_recoveryRequester: STRING;
	m_recoveryState: ERecoveryState;
	m_recoverySequence: LinearSequence;
	m_tonStrategyReceivedTimeout: TON;
	m_alarmId: UINT := 0;
	
	m_finishedAutonomously: ARRAY [ResiConst.ARR_MIN..ResiConst.BEHAVIORS_ARR_MAX] OF BOOL;
	m_finishedAutoBuffer: ARRAY [ResiConst.ARR_MIN..ResiConst.BEHAVIORS_ARR_MAX] OF BOOL;
	
	(* ABORT *)
	m_abortState: EAbortState;
	
	(* RUNTIME EXPRESSIONS, CONDITIONS *)
	m_boolExpressions: ARRAY [ResiConst.ARR_MIN..ResiConst.RT_EXPRS_MAX] OF BoolExpression(0, EBoolOperation.none, 0);
	
	// CUSTOM STRATEGY
	m_stepReaders: 	ARRAY [ResiConst.ARR_MIN..ResiConst.MAX_SYNC_PARTNERS] OF 
					ARRAY [ResiConst.ARR_MIN..ResiConst.STRAT_LEN_MAX] OF ADSREADEX;
	m_stepWriters: 	ARRAY [ResiConst.ARR_MIN..ResiConst.MAX_SYNC_PARTNERS] OF 
					ARRAY [ResiConst.ARR_MIN..ResiConst.STRAT_LEN_MAX] OF ADSWRITE;
	m_stepStates: 	ARRAY [ResiConst.ARR_MIN..ResiConst.MAX_SYNC_PARTNERS] OF 
					ARRAY [ResiConst.ARR_MIN..ResiConst.STRAT_LEN_MAX] OF EOperationResult;
	m_busyState:	EOperationResult := EOperationResult.busy;
	m_anyBusy: 		BOOL;
END_VAR

PROPERTY AbortActive : BOOL
GET
AbortActive := m_abortState = EAbortState.requested OR m_abortState = EAbortState.aborting;
END_GET
END_PROPERTY

METHOD AddPrimitive : BOOL
VAR_INPUT
	i_ptrPrimitive: POINTER TO ControlPrimitiveBase;
END_VAR
IF m_ptrPrimitives[i_ptrPrimitive^.Id] <> 0 THEN
	// already initialized a primitive with that ID
	AddPrimitive := FALSE;
	RETURN;
END_IF

m_ptrPrimitives[i_ptrPrimitive^.Id] := i_ptrPrimitive;
AddPrimitive := TRUE;
END_METHOD

METHOD AddSequence : BOOL
VAR_INPUT
	i_ptrSequence: POINTER TO ModuleSequenceBase;
END_VAR
IF m_ptrSequences[i_ptrSequence^.Id] <> 0 THEN
	// already initialized a sequence with that ID
	AddSequence := FALSE;
	RETURN;
END_IF

m_ptrSequences[i_ptrSequence^.Id] := i_ptrSequence;
AddSequence := TRUE;
END_METHOD

(* Applies a new compensation, i.e., the replacement of a "sick" primitive with another primitive or  a module sequence. *)
METHOD Compensate : BOOL
VAR_INPUT
	i_ptrCompensation: POINTER TO SCompensation;
END_VAR
IF i_ptrCompensation^.NewType = EBehaviorType.none THEN
	Compensate := FALSE;
	RETURN;
END_IF

CASE i_ptrCompensation^.NewType OF
	EBehaviorType.control_primitive:
		// check if the specified replacement exists
		IF m_ptrPrimitives[i_ptrCompensation^.NewId] = 0 THEN
			Compensate := FALSE;
			RETURN;
		END_IF
		
		m_retargets[i_ptrCompensation^.SickPrimitiveId].RetargetType := ERetargetType.primitive_target;
		m_retargets[i_ptrCompensation^.SickPrimitiveId].TargetId := i_ptrCompensation^.NewId;
		m_retargets[i_ptrCompensation^.SickPrimitiveId].OverwriteParams := i_ptrCompensation^.ParameterSets[0];

	EBehaviorType.user_sequence:
		// check if the specified replacement exists
		IF m_ptrSequences[i_ptrCompensation^.NewId] = 0 THEN
			Compensate := FALSE;
			RETURN;
		END_IF
		
		m_retargets[i_ptrCompensation^.SickPrimitiveId].RetargetType := ERetargetType.sequence_target;
		m_retargets[i_ptrCompensation^.SickPrimitiveId].TargetId := i_ptrCompensation^.NewId;
		m_retargets[i_ptrCompensation^.SickPrimitiveId].OverwriteParams := i_ptrCompensation^.ParameterSets[0];

	EBehaviorType.generated_sequence:
		m_compSeqs[m_compSeqsIdx].ProvideServices(THIS, THIS^.m_ptrStateTracker);
		m_compSeqs[m_compSeqsIdx].i_primitiveParams := i_ptrCompensation^.ParameterSets;
		m_compSeqs[m_compSeqsIdx].i_primitiveIds := i_ptrCompensation^.PrimitiveIds;
		
		m_ptrSequences[m_compSeqsIdx] := ADR(m_compSeqs[m_compSeqsIdx]);
		m_retargets[i_ptrCompensation^.SickPrimitiveId].RetargetType := ERetargetType.sequence_target;
		m_retargets[i_ptrCompensation^.SickPrimitiveId].TargetId := m_compSeqsIdx;
		
		m_compSeqsIdx := m_compSeqsIdx + 1;
END_CASE

Compensate := TRUE;
END_METHOD

PROPERTY CustomStrategyReady : BOOL
GET
CustomStrategyReady := THIS^.raIn_customStrategy.State = EStrategyStates.ready;
END_GET
END_PROPERTY

METHOD CyclicManageBehavior : BOOL
VAR CONSTANT
	TIMEOUT: TIME := T#10S;
END_VAR
VAR
	i: UINT;
	p_id: UINT;
	
	m_sequenceStatus: EOperationResult;
	m_allAborted: BOOL;
	
	m_valExpr: IValExp;
	m_recoveryRes: EOperationResult;
	m_emptyRecovery: SRecovery;
	m_emptyParams: ParameterSet;
	
	m_tmpExpr: IExpression;
END_VAR
// ABORT
CASE m_abortState OF
	EAbortState.none:
		;
		
	EAbortState.requested:
		m_abortState := EAbortState.aborting;
		
	EAbortState.aborting:
		m_allAborted := TRUE;
		FOR i := ResiConst.ARR_MIN TO ResiConst.BEHAVIORS_ARR_MAX DO
			IF m_ptrPrimitives[i] <> 0 THEN
				IF NOT m_ptrPrimitives[i]^.Abort() THEN
					m_allAborted := FALSE;
				END_IF
			END_IF	
		END_FOR
		
		IF m_allAborted THEN
			m_abortState := EAbortState.aborted;
		END_IF
		
	EAbortState.aborted:
		m_abortState := EAbortState.none;
END_CASE

// COMPENSATION
FOR i := ResiConst.ARR_MIN TO ResiConst.COMPENSATIONS_ARR_MAX DO
	IF raIn_compensations[i].IsActive THEN
		CONTINUE;
	END_IF
	
	raIn_compensations[i].IsActive := Compensate(ADR(raIn_compensations[i])); 
END_FOR

// while a compensation sequence is active, other primitives must be suspended to avoid interference (handled at MAIN level)
CASE m_activeCompensationState OF
	ECompSeqState.preparing:
		// finish all running primitives
		IF FinishPrimitives(i_abortRecoveries := TRUE) THEN
			m_activeCompensationState := ECompSeqState.running;
			
			// Reset the "finished autonomously" flag for all primitives involved in this compensation. Otherwise, the Execute 
			// method will return TRUE without doing anything.
			m_finishedAutoBuffer := m_finishedAutonomously;
			FOR i := ResiConst.ARR_MIN TO ResiConst.MODULE_SEQ_ARR_MAX DO
				p_id := m_compSeqs[m_activeCompensationIdx].i_primitiveIds[i];
				m_finishedAutonomously[p_id] := FALSE;
			END_FOR
		END_IF
	
	ECompSeqState.running:
		m_ptrSequences[m_activeCompensationIdx]^(o_status => m_sequenceStatus);
		IF m_sequenceStatus = EOperationResult.success THEN
			m_activeCompensationState := ECompSeqState.finished;
		END_IF
		
	ECompSeqState.finished:
		// restore the "finished autonomously" flags again
		m_finishedAutonomously := m_finishedAutoBuffer;	
		m_activeCompensationState := ECompSeqState.none;
END_CASE

// RECOVERY, DEFINITION
CASE m_recoveryState OF
	ERecoveryState.requested:
		m_tonStrategyReceivedTimeout(IN := FALSE);
		
		IF m_alarmId = 0 THEN
			// if the requested state is a ValueExpression, it's a request for definition
			IF __QUERYINTERFACE(m_conditionToRecover, m_valExpr) THEN
				m_alarmId := ESpecialAlarmIds.definition_request;
			ELSE
				m_alarmId := ESpecialAlarmIds.recovery_request;
			END_IF
			
			m_ptrErrorMgr^.AddMessage(
				i_alarmId := m_alarmId,
				i_active := TRUE,
				i_severity := ESeverity.warning,
				i_instanceName := m_recoveryRequester);
		END_IF

		// TODO - unify approaches!
		// in the AT-Symp setup, recoveries are handled by modifying the custom strategy
		m_recoveryState := ERecoveryState.none;
		raOut_recoveryRequest.ChangeTrigger := raOut_recoveryRequest.ChangeTrigger + 1;
		raOut_recoveryRequest.RequestedState := m_conditionToRecover.ToString();
		m_alarmId := 0;
			
// 		// finish all running primitives safely before recovery
// 		IF FinishPrimitives(i_abortRecoveries := FALSE) THEN
// 			raOut_recoveryRequest.ChangeTrigger := raOut_recoveryRequest.ChangeTrigger + 1;
// 			raOut_recoveryRequest.RequestedState := m_conditionToRecover.ToString();
// 			m_alarmId := 0;
// 			
// 			m_recoveryState := ERecoveryState.awaiting;
// 		END_IF
		
	ERecoveryState.awaiting:
		m_tonStrategyReceivedTimeout(IN := TRUE, PT := TIMEOUT);
		IF m_tonStrategyReceivedTimeout.Q THEN
			m_recoveryState := ERecoveryState.failed; 
		ELSIF raIn_recoveryAvailable THEN
			m_recoveryState := ERecoveryState.running;
		END_IF
		
	// the state is only "failed" if the CPA cannot deliver any viable strategy
	ERecoveryState.failed:
		m_recoveryState := ERecoveryState.none;
		raOut_recoveryRequest.RequestedState := '';
		
	ERecoveryState.running:
		m_recoverySequence(
			i_params := raIn_Recovery.RecoveryParameters,
			i_primitiveIds := raIn_Recovery.RecoveryStrategy,
			o_status => m_recoveryRes);
		
		// if unsuccessful, the respective primitive has already requested a new recovery
		IF m_recoveryRes = EOperationResult.success THEN
			m_recoveryState := ERecoveryState.completed;
		END_IF
		
	ERecoveryState.completed:
		m_recoveryState := ERecoveryState.none;
		
		// reset
		raIn_recovery := m_emptyRecovery;
		raIn_recoveryAvailable := FALSE;
END_CASE

// EDITABLE CONDITIONS
FOR i := ResiConst.ARR_MIN TO ResiConst.COMPENSATIONS_ARR_MAX DO
	IF raIn_runtimeConditions[i].ExpressionType <> EExpressionType.none AND NOT raIn_runtimeConditions[i].IsActive THEN
		m_tmpExpr := GetExpression(
			raIn_runtimeConditions[i].ExpressionType, 
			raIn_runtimeConditions[i].ExpressionIdx);
		
		SetPrimitiveCondition(
			raIn_runtimeConditions[i].PrimitiveId, 
			raIn_runtimeConditions[i].IsPre,
			m_tmpExpr);
		
		raIn_runtimeConditions[i].IsActive := TRUE;
	END_IF
	IF raIn_runtimeInterlocks[i].ExpressionType <> EExpressionType.none AND NOT raIn_runtimeInterlocks[i].IsActive THEN
		m_tmpExpr := GetExpression(
			raIn_runtimeInterlocks[i].ExpressionType, 
			raIn_runtimeInterlocks[i].ExpressionIdx);
			
		m_ptrStateTracker^.AddInterlock(m_tmpExpr, raIn_runtimeInterlocks[i].DefaultValue);
		raIn_runtimeInterlocks[i].IsActive := TRUE;
	END_IF
END_FOR

// CP STATUS: keep executing all "successful" primitives until their status returns to "none"
FOR i := ResiConst.ARR_MIN TO ResiConst.BEHAVIORS_ARR_MAX DO
	IF m_ptrPrimitives[i] <> 0 THEN
		IF m_ptrPrimitives[i]^.o_status = EOperationResult.success THEN
			Execute(EBehaviorType.control_primitive, i, m_emptyParams);
		END_IF
	END_IF
END_FOR
END_METHOD

(* Executes the requested Control Primitive or Module Sequence. 
COMPENSATION: If a compensation was previously registered, the replacement is executed instead. *)
METHOD Execute : EOperationResult
VAR_INPUT
	i_type: EBehaviorType;
	i_id: UINT;
	i_params: ParameterSet;
END_VAR
VAR
	i: UINT;
	m_actualId: UINT;
	m_result: INT;
	m_overwrites: ARRAY [ResiConst.ARR_MIN..ResiConst.PARAMS_ARR_MAX] OF SNamedValue;
	m_prevStatus: EOperationResult;
END_VAR
// set/overwrite additional parameters specified by the retargeting
IF m_retargets[i_id].RetargetType <> ERetargetType.not_retargeted THEN
	i_params := i_params;
	m_overwrites := m_retargets[i_id].OverwriteParams.Parameters;
	FOR i := ResiConst.ARR_MIN TO ResiConst.PARAMS_ARR_MAX DO
		IF m_overwrites[i].DataType = EDataType.binary THEN
			i_params.SetParam_Binary(m_overwrites[i].Name, m_overwrites[i].Value.Binary);
		ELSIF m_overwrites[i].DataType = EDataType.numeric THEN
			i_params.SetParam_Numeric(m_overwrites[i].Name, m_overwrites[i].Value.Numeric);
		ELSIF m_overwrites[i].DataType = EDataType.string_t THEN
			i_params.SetParam_String(m_overwrites[i].Name, m_overwrites[i].Value.String_t);
		END_IF
	END_FOR	
END_IF

IF i_type = EBehaviorType.control_primitive THEN
	// if the primitive was finished in the background before recovery (FinishPrimitives), return the success signal
	IF m_finishedAutonomously[i_id] THEN
		Execute := EOperationResult.success;
		m_finishedAutonomously[i_id] := FALSE;
		RETURN;
	END_IF	

	CASE m_retargets[i_id].RetargetType OF
		// execute the requested Control Primitive
		ERetargetType.not_retargeted:
			IF m_ptrPrimitives[i_id] = 0 THEN
				Execute := EOperationResult.failed;
				RETURN;
			END_IF
			
			m_prevStatus := m_ptrPrimitives[i_id]^.o_status;
			m_ptrPrimitives[i_id]^(
				i_params := i_params,
				o_status => Execute);
			
			// CP-Base state machine always returns None on first call -> messes up the logic sometimes...
			IF m_prevStatus = EOperationResult.none AND m_ptrPrimitives[i_id]^.o_status = EOperationResult.none THEN
				Execute := EOperationResult.waiting;
			END_IF
			
		// primitive compensated by other primitive
		ERetargetType.primitive_target:
			IF m_ptrPrimitives[m_retargets[i_id].TargetId] = 0 THEN
				Execute := EOperationResult.failed;
				RETURN;
			END_IF
			
			m_ptrPrimitives[m_retargets[i_id].TargetId]^(
				i_params := i_params,
				o_status => Execute);
			
		// primitive compensated by sequence (i_primitiveParams were already parsed in ProcessManager.Compensate())
		ERetargetType.sequence_target:
			IF m_ptrSequences[m_retargets[i_id].TargetId] = 0 THEN
				Execute := EOperationResult.failed;
				RETURN;
			END_IF
			
			// the rest is handled in CyclicManageBehavior
			m_activeCompensationState := ECompSeqState.preparing;
			m_activeCompensationIdx := m_retargets[i_id].TargetId;
			Execute := EOperationResult.success;
	END_CASE

ELSIF i_type = EBehaviorType.user_sequence THEN
	// execute the requested Module Sequence
	IF m_ptrSequences[i_id] = 0 THEN
		Execute := EOperationResult.failed;
		RETURN;
	END_IF
	
	m_ptrSequences[i_id]^(
		i_params := i_params,
		o_status => Execute);
		
ELSE 
	// generated_sequence cannot be called directly
	Execute := EOperationResult.failed;
END_IF
END_METHOD

METHOD ExecuteCustomStrategy : EOperationResult
VAR
	startInit: BOOL;
	allSucceeded: BOOL;
	
	i: INT;
	ui: UINT;
	
	stepIdx: UINT;
	transIdx: UINT;
	
	step: SStep;
	cp_status: EOperationResult;
	trans: STransition;
	expr: IExpression;
	
	prevStepIdx: INT;
	nextStepIdx: INT;
END_VAR
// STRATEGY STATES
CASE raIn_customStrategy.State OF
	EStrategyStates.ready:
		raIn_customStrategy.State := EStrategyStates.running;
		m_ptrErrorMgr^.AddMessage(ESpecialAlarmIds.strategy_received, TRUE, ESeverity.info, 'ProcessManager');
		RETURN;
		
	EStrategyStates.running:
		ExecuteCustomStrategy := EOperationResult.busy;
	
	EStrategyStates.halting:
		IF NOT m_anyBusy THEN
			raIn_customStrategy.State := EStrategyStates.halted;
		END_IF
		RETURN;
		
	EStrategyStates.done:
		ExecuteCustomStrategy := EOperationResult.success;
		RETURN;
		
	ELSE
		ExecuteCustomStrategy := EOperationResult.none;
		RETURN;
END_CASE


// STEP EXECUTION
FOR stepIdx := ResiConst.ARR_MIN TO ResiConst.STRAT_LEN_MAX DO
	step := raIn_customStrategy.Steps[stepIdx];
	IF m_ptrPrimitives[step.BehaviorId] = 0 THEN
		CONTINUE;
	END_IF
	
	IF step.State = EOperationResult.busy THEN
		// NOTE: currently, only success/failure/busy/recovering are differentiated for steps
		cp_status := Execute(step.BehaviorType, step.BehaviorId, step.Parameters);
		IF cp_status = EOperationResult.busy OR cp_status = EOperationResult.waiting THEN
			step.State := EOperationResult.busy;
		ELSE
			// success, revocering, failed
			step.State := cp_status;
		END_IF
	ELSIF step.State = EOperationResult.recovering THEN
		// keep executing until the status changes
		step.State := Execute(step.BehaviorType, step.BehaviorId, step.Parameters);
	END_IF
	
	raIn_customStrategy.Steps[stepIdx] := step;
END_FOR

IF NOT raIn_customStrategy.IsMaster THEN
	RETURN;
END_IF


// ##### MASTER REGION: COORDINATE EXECUTION #####
// ############ EXECUTE ACTIVE STEPS #############
startInit := TRUE;
m_anyBusy := FALSE;
FOR stepIdx := ResiConst.ARR_MIN TO ResiConst.STRAT_LEN_MAX DO
	step := raIn_customStrategy.Steps[stepIdx];
	CASE step.State OF
		EOperationResult.none:
			;
		
		EOperationResult.waiting:
			startInit := FALSE;
			m_anyBusy := TRUE;
			IF stepIdx = INT_TO_UINT(ESpecialStepIds.end) THEN
				step.State := EOperationResult.none;
				IF raIn_customStrategy.LoopStrategy THEN
					startInit := TRUE;
				ELSE
					raIn_customStrategy.State := EStrategyStates.done;
					RETURN;
				END_IF
			ELSIF step.BehaviorType = EBehaviorType.none THEN
				// if no behavior is needed, the step is immediately considered as succeeded
				step.State := EOperationResult.success;
			ELSE
				step.State := EOperationResult.busy;
			END_IF
			
		EOperationResult.busy:
			startInit := FALSE;
			m_anyBusy := TRUE;
			IF m_ptrPrimitives[step.BehaviorId] = 0 THEN
				// instruct another PLC to execute
				m_stepWriters[step.ExecutorIdx][stepIdx](
					NETID := step.ExtSymbols[step.ExecutorIdx].NetId,
					PORT := step.ExtSymbols[step.ExecutorIdx].Port,
					IDXGRP := step.ExtSymbols[step.ExecutorIdx].IdxGrp,
					IDXOFFS := step.ExtSymbols[step.ExecutorIdx].IdxOffs,
					LEN := SIZEOF(m_busyState),
					SRCADDR := ADR(m_busyState),
					WRITE := TRUE);
				
				// flush a potentially buffered old "success" result
				m_stepReaders[step.ExecutorIdx][stepIdx](READ := FALSE);
				m_stepReaders[step.ExecutorIdx][stepIdx](
					NETID := step.ExtSymbols[step.ExecutorIdx].NetId,
					PORT := step.ExtSymbols[step.ExecutorIdx].Port,
					IDXGRP := step.ExtSymbols[step.ExecutorIdx].IdxGrp,
					IDXOFFS := step.ExtSymbols[step.ExecutorIdx].IdxOffs,
					LEN := SIZEOF(m_stepStates[step.ExecutorIdx][stepIdx]),
					DESTADDR := ADR(m_stepStates[step.ExecutorIdx][stepIdx]),
					READ := TRUE);
				
				IF m_stepStates[step.ExecutorIdx][stepIdx] = m_busyState THEN
					m_stepWriters[step.ExecutorIdx][stepIdx](WRITE := FALSE);
					step.State := EOperationResult.success;
				END_IF
			END_IF
			
		EOperationResult.success:
			startInit := FALSE;
			IF step.BehaviorType <> EBehaviorType.none AND m_ptrPrimitives[step.BehaviorId] = 0 THEN
				// wait until external state returns success
				m_stepReaders[step.ExecutorIdx][stepIdx](READ := FALSE);
				m_stepReaders[step.ExecutorIdx][stepIdx](
					NETID := step.ExtSymbols[step.ExecutorIdx].NetId,
					PORT := step.ExtSymbols[step.ExecutorIdx].Port,
					IDXGRP := step.ExtSymbols[step.ExecutorIdx].IdxGrp,
					IDXOFFS := step.ExtSymbols[step.ExecutorIdx].IdxOffs,
					LEN := SIZEOF(m_stepStates[step.ExecutorIdx][stepIdx]),
					DESTADDR := ADR(m_stepStates[step.ExecutorIdx][stepIdx]),
					READ := TRUE);
				IF m_stepStates[step.ExecutorIdx][stepIdx] = EOperationResult.success THEN
					step.State := EOperationResult.synced_success;
				ELSIF m_stepStates[step.ExecutorIdx][stepIdx] = EOperationResult.failed THEN
					step.State := EOperationResult.failed;
				ELSIF m_stepStates[step.ExecutorIdx][stepIdx] = EOperationResult.recovering THEN
					step.State := EOperationResult.recovering;
				ELSE
					// don't store external state in the step struct because it will screw with this state machine
					m_anyBusy := TRUE;
				END_IF
			ELSE
				step.State := EOperationResult.synced_success;
			END_IF
		
		EOperationResult.synced_success:
			startInit := FALSE;
			
		EOperationResult.failed:
			startInit := FALSE;
			allSucceeded := FALSE;
			ExecuteCustomStrategy := EOperationResult.failed;
			RETURN;
		
		EOperationResult.recovering:
			raIn_customStrategy.State := EStrategyStates.halting;
			m_ptrErrorMgr^.AddMessage(ESpecialAlarmIds.recovery_request, TRUE, ESeverity.info, 'ProcessManager');
	END_CASE
	
	raIn_customStrategy.Steps[stepIdx] := step;
END_FOR

IF raIn_customStrategy.State = EStrategyStates.halting THEN
	// wait for all steps to finish; don't start new ones below
	RETURN;
END_IF

IF startInit THEN
	// start the initial step
	step := raIn_customStrategy.Steps[ESpecialStepIds.start];
	step.State := EOperationResult.waiting;
	raIn_customStrategy.Steps[ESpecialStepIds.start] := step;
END_IF


// ###### AWAIT AND FIRE TRANSITIONS ######
FOR transIdx := ResiConst.ARR_MIN TO ResiConst.STRAT_LEN_MAX DO
	trans := raIn_customStrategy.Transitions[transIdx];
	IF NOT trans.IsSet THEN
		CONTINUE;
	END_IF
	
	// 1) all previous steps must have succeeded (NOTE: this is different from the SFC language)
	allSucceeded := TRUE;
	FOR ui := ResiConst.ARR_MIN TO ResiConst.STRAT_PARALLEL_MAX DO
		prevStepIdx := trans.PrevStepIds[ui];
		IF prevStepIdx = ESpecialStepIds.unset THEN
			CONTINUE;
		END_IF
		
		step := raIn_customStrategy.Steps[prevStepIdx];
		IF step.State <> EOperationResult.synced_success THEN
			allSucceeded := FALSE;
			EXIT;
		END_IF
	END_FOR
	
	IF NOT allSucceeded THEN
		CONTINUE;
	END_IF

	// 2) wait for the transition's own condition to become TRUE
	expr := GetExpression(trans.ExpressionType, trans.ExpressionIdx);
	IF expr.IsTrue(m_ptrStateTracker^.PtrProcessState) THEN
		// switch the previous steps to "none" and next ones to "waiting"
		FOR ui := ResiConst.ARR_MIN TO ResiConst.STRAT_PARALLEL_MAX DO
			prevStepIdx := trans.PrevStepIds[ui];
			IF prevStepIdx <> ESpecialStepIds.unset THEN
				step := raIn_customStrategy.Steps[prevStepIdx];
				step.State := EOperationResult.none;
				raIn_customStrategy.Steps[prevStepIdx] := step;
			END_IF
			
			nextStepIdx := trans.NextStepIds[ui];
			IF nextStepIdx <> ESpecialStepIds.unset THEN
				step := raIn_customStrategy.Steps[nextStepIdx];
				step.State := EOperationResult.waiting;
				raIn_customStrategy.Steps[nextStepIdx] := step;
			END_IF
		END_FOR
	END_IF
END_FOR
END_METHOD

// When a compensation *sequence* is active, other primitive calls must be suspended to avoid interference.
PROPERTY FaultHandlingActive : BOOL
GET
FaultHandlingActive := m_activeCompensationState = ECompSeqState.preparing 
	OR m_activeCompensationState = ECompSeqState.running
	OR m_recoveryState = ERecoveryState.requested
	OR m_recoveryState = ERecoveryState.awaiting
	OR m_recoveryState = ERecoveryState.running;
END_GET
END_PROPERTY

PROPERTY FaultHandlingFailed : BOOL
GET
FaultHandlingFailed := m_recoveryState = ERecoveryState.failed;
END_GET
END_PROPERTY

METHOD FB_init : BOOL
VAR_INPUT
	bInitRetains : BOOL; // if TRUE, the retain variables are initialized (warm start / cold start)
	bInCopyCode : BOOL;  // if TRUE, the instance afterwards gets moved into the copy code (online change)
END_VAR
VAR
	i: UINT;
	j: UINT;
END_VAR
// reset the strategy transitions
FOR i := ResiConst.ARR_MIN TO ResiConst.STRAT_LEN_MAX DO
	FOR j := ResiConst.ARR_MIN TO ResiConst.STRAT_PARALLEL_MAX DO
		raIn_customStrategy.Transitions[i].PrevStepIds[j] := -1;
		raIn_customStrategy.Transitions[i].NextStepIds[j] := -1;
	END_FOR
END_FOR
END_METHOD

METHOD FinishPrimitives : BOOL
VAR_INPUT
	i_abortRecoveries: BOOL;
END_VAR
VAR
	i: UINT;
	m_allFinished: BOOL;
END_VAR
m_allFinished := TRUE;
FOR i := ResiConst.ARR_MIN TO ResiConst.BEHAVIORS_ARR_MAX DO
	IF m_ptrPrimitives[i] <> 0 THEN
		IF m_ptrPrimitives[i]^.o_status = EOperationResult.busy 
			OR m_ptrPrimitives[i]^.o_status = EOperationResult.waiting 
			OR (i_abortRecoveries AND m_ptrPrimitives[i]^.o_status = EOperationResult.recovering) THEN
			
			m_ptrPrimitives[i]^();
			m_allFinished := FALSE;
			
			IF m_ptrPrimitives[i]^.o_status = EOperationResult.success THEN
				// after finishing, the success must be communicated to the application code once the automatic operation resumes (after recovery)
				m_finishedAutonomously[i] := TRUE;
			END_IF
		END_IF
	END_IF	
END_FOR

FinishPrimitives := m_allFinished;
END_METHOD

METHOD GetBehaviorPtr : POINTER TO BehaviorBase
VAR_INPUT
	i_type: EBehaviorType;
	i_id: UINT;
END_VAR
IF i_type = EBehaviorType.control_primitive THEN
	GetBehaviorPtr := m_ptrPrimitives[i_id];
ELSIF i_type = EBehaviorType.user_sequence OR i_type = EBehaviorType.generated_sequence THEN
	GetBehaviorPtr := m_ptrSequences[i_id];
ELSE
	GetBehaviorPtr := 0;
END_IF
END_METHOD

METHOD GetExpression : IExpression
VAR_INPUT
	i_type: EExpressionType;
	i_idx: UINT;
END_VAR
CASE i_type OF
	EExpressionType.boolean:
		THIS^.m_boolExpressions[i_idx].FB_init(
			FALSE, FALSE,
			i_left := THIS^.GetExpression(raIn_boolExprSpecs[i_idx].LeftType, raIn_boolExprSpecs[i_idx].LeftIdx),
			i_sign := raIn_boolExprSpecs[i_idx].Operator,
			i_right := THIS^.GetExpression(raIn_boolExprSpecs[i_idx].RightType, raIn_boolExprSpecs[i_idx].RightIdx));
		GetExpression := THIS^.m_boolExpressions[i_idx];
	
	EExpressionType.comparison:
		GetExpression := raIn_compExpressions[i_idx];
	
	EExpressionType.value:
		GetExpression := raIn_valueExpressions[i_idx];
	
	ELSE
		GetExpression := 0;
END_CASE
END_METHOD

METHOD ProvideServices : BOOL
VAR_INPUT
	i_ptrStateTracker: POINTER TO StateTracker;
	i_ptrErrorMgr: POINTER TO ErrorManagerBase;
END_VAR
THIS^.m_ptrStateTracker := i_ptrStateTracker;
THIS^.m_ptrErrorMgr := i_ptrErrorMgr;

THIS^.m_recoverySequence.ProvideServices(THIS, i_ptrStateTracker);
END_METHOD

METHOD RequestAbort : BOOL
VAR_INPUT
END_VAR
IF m_abortState = EAbortState.none THEN
	m_abortState := EAbortState.requested;
END_IF
END_METHOD

METHOD RequestRecovery : BOOL
VAR_INPUT
	i_desiredState: IExpression;
	i_senderName: STRING;
END_VAR
// "recursive" recoveries are not supported
IF m_recoveryState <> ERecoveryState.none THEN
	RETURN;
END_IF

m_recoveryState := ERecoveryState.requested;
m_conditionToRecover := i_desiredState;
m_recoveryRequester := i_senderName;
END_METHOD

METHOD ResetConfiguration : BOOL
VAR
	i: UINT;
	emptyVal: ValueExpression(EDataType.none, FALSE, 0, '', FALSE);
	emptyCpr: ComparisonExpression(0, EComparisonType.none, EDataType.none, FALSE, 0, '', FALSE);
	emptyBool: BoolExpression(0, EBoolOperation.none, 0);
	emptyBoolS: SBoolExpressionSpec;
	emptyNums: ARRAY [ResiConst.ARR_MIN..ResiConst.MODULE_SEQ_ARR_MAX] OF UINT;
	emptyCond: SPrimitiveCondition;
	emptyItl: SInterlock;
	emptyStep: SStep;
	emptyTrans: STransition;
END_VAR
FOR i := ResiConst.ARR_MIN TO ResiConst.COMPENSATIONS_ARR_MAX DO
	raIn_compensations[i].IsActive := FALSE;
	raIn_compensations[i].NewId := 0;
	raIn_compensations[i].NewType := EBehaviorType.none;
	raIn_compensations[i].SickPrimitiveId := 0;
	// TODO - reset all the arrays too?
END_FOR

raOut_recoveryRequest.RequestedState := '';
raIn_recoveryAvailable := FALSE;
raIn_recovery.RecoveryParameters.Reset();
raIn_recovery.RecoveryStrategy := emptyNums;

FOR i := ResiConst.ARR_MIN TO ResiConst.RT_EXPRS_MAX DO
	raIn_valueExpressions[i] := emptyVal;
	raIn_compExpressions[i] := emptyCpr;
	raIn_boolExprSpecs[i] := emptyBoolS;
	m_boolExpressions[i] := emptyBool;
END_FOR

FOR i := ResiConst.ARR_MIN TO ResiConst.COMPENSATIONS_ARR_MAX DO
	raIn_runtimeConditions[i] := emptyCond;
	raIn_runtimeInterlocks[i] := emptyItl;
END_FOR

raIn_customStrategy.State := EStrategyStates.none;
raIn_customStrategy.LoopStrategy := FALSE;
raIn_customStrategy.IsMaster := FALSE;
raIn_customStrategy.NumPartners := 0;
FOR i := ResiConst.ARR_MIN TO ResiConst.STRAT_LEN_MAX DO
	raIn_customStrategy.Steps[i] := emptyStep;
	raIn_customStrategy.Transitions[i] := emptyTrans;
END_FOR
END_METHOD

METHOD SetAllConditionsTrue : BOOL
VAR
	i: UINT;
END_VAR
FOR i := ResiConst.ARR_MIN TO ResiConst.BEHAVIORS_ARR_MAX DO
	IF m_ptrPrimitives[i] <> 0 THEN
		m_ptrPrimitives[i]^.Precondition := m_trueValue;
		m_ptrPrimitives[i]^.Postcondition := m_trueValue;
	END_IF
END_FOR
END_METHOD

METHOD SetPrimitiveCondition : BOOL
VAR_INPUT
	i_primitiveId: UINT;
	i_isPre: BOOL;
	i_condition: IExpression;
END_VAR
IF i_isPre THEN
	THIS^.m_ptrPrimitives[i_primitiveId]^.Precondition := i_condition;
ELSE
	THIS^.m_ptrPrimitives[i_primitiveId]^.Postcondition := i_condition;
END_IF
END_METHOD

END_FUNCTION_BLOCK

// ---- Models/ProcessState/ProcessCondition/ValueExpression.TcPOU
{attribute 'OPC.UA.DA.StructuredType' := '1'}
FUNCTION_BLOCK ValueExpression IMPLEMENTS IExpression, IValExp
VAR_OUTPUT
	o_value: SValue;
END_VAR

METHOD FB_init : BOOL
VAR_INPUT
	bInitRetains : BOOL; // if TRUE, the retain variables are initialized (warm start / cold start)
	bInCopyCode : BOOL;  // if TRUE, the instance afterwards gets moved into the copy code (online change)
	
	i_dataType: EDataType;
	i_binaryValue: BOOL;
	i_numericValue: LREAL;
	i_stringValue: STRING;
	i_defined: BOOL;
END_VAR
o_value.DataType := i_dataType;
o_value.Defined := i_defined;

CASE i_dataType OF
	EDataType.binary:
		o_value.Value.Binary := i_binaryValue;

	EDataType.numeric:
		o_value.Value.Numeric := i_numericValue;
		
	EDataType.string_t:
		o_value.Value.String_t := i_stringValue;
END_CASE
END_METHOD

METHOD IsTrue : BOOL
VAR_INPUT
	i_ptrProcessState: POINTER TO ProcessState;
END_VAR
IsTrue := o_value.DataType = EDataType.binary AND o_value.Value.Binary;
END_METHOD

METHOD ToString : STRING(256)
VAR_INPUT
END_VAR
CASE o_value.DataType OF
	EDataType.binary:
		ToString := TO_STRING(o_value.Value.Binary);
		
	EDataType.numeric:
		ToString := TO_STRING(o_value.Value.Numeric);
		
	EDataType.string_t:
		ToString := o_value.Value.String_t;
	
	ELSE
		ToString := '';
END_CASE
END_METHOD

END_FUNCTION_BLOCK

// ---- Models/ProcessState/ProcessState.TcPOU
FUNCTION_BLOCK ProcessState
VAR_INPUT
END_VAR
VAR_OUTPUT
END_VAR
VAR
	m_ptrProcMgr: POINTER TO ProcessManager;
	m_values: ARRAY [ResiConst.ARR_MIN..ResiConst.STATE_ARR_MAX] OF SValue;
	m_varExp: ValueExpression(EDataType.numeric, FALSE, 0, '', TRUE);
END_VAR

// manages all the system variables

METHOD ProvideServices : BOOL
VAR_INPUT
	i_ptrProcMgr: POINTER TO ProcessManager;
END_VAR
m_ptrProcMgr := i_ptrProcMgr;
END_METHOD

METHOD Retrieve : SValue
VAR_INPUT
	i_id: UINT;
	i_checkDef: BOOL;
END_VAR
VAR
	m_val: SValue;
END_VAR
m_val := m_values[i_id];

IF i_checkDef THEN
	IF m_val.Defined THEN
		Retrieve:= m_val;
	ELSE
		m_varExp.FB_init(FALSE, FALSE, EDataType.numeric, FALSE, i_id, '', TRUE);
		THIS^.m_ptrProcMgr^.RequestRecovery(m_varExp, 'ProcessState.Retrieve');
	END_IF	
ELSE
	Retrieve := m_val;
END_IF
END_METHOD

METHOD SetValue : BOOL
VAR_INPUT
	i_id: UINT;
	i_val: SValue;
END_VAR
SetValue := FALSE;
m_values[i_id].DataType := i_val.DataType;
m_values[i_id].Defined := i_val.Defined;

CASE i_val.DataType OF
	EDataType.binary:
		m_values[i_id].Value.Binary := i_val.Value.Binary;
		SetValue := TRUE;
		
	EDataType.numeric:
		m_values[i_id].Value.Numeric := i_val.Value.Numeric;
		SetValue := TRUE;
		
	EDataType.string_t:
		m_values[i_id].Value.String_t := i_val.Value.String_t;
		SetValue := TRUE;
END_CASE
END_METHOD

METHOD UpdateState_Binary : BOOL
VAR_INPUT
	i_id: UINT;
	i_value: BOOL;
	
	// writes even if the existing data type does not match
	i_force: BOOL;
END_VAR
IF i_force THEN
	m_values[i_id].DataType := EDataType.binary;
	m_values[i_id].Value.Binary := FALSE;
END_IF

IF m_values[i_id].DataType = EDataType.binary THEN
	m_values[i_id].Value.Binary := i_value;
	UpdateState_Binary := TRUE;
ELSE
	UpdateState_Binary := FALSE;
END_IF
END_METHOD

METHOD UpdateState_Defined : BOOL
VAR_INPUT
	i_id: UINT;
	i_defined: BOOL;
END_VAR
m_values[i_id].Defined := i_defined;
UpdateState_Defined := TRUE;
END_METHOD

METHOD UpdateState_Numeric : BOOL
VAR_INPUT
	i_id: UINT;
	i_value: LREAL;
	
	// writes even if the existing data type does not match
	i_force: BOOL;
END_VAR
IF i_force THEN
	m_values[i_id].DataType := EDataType.numeric;
	m_values[i_id].Value.Numeric := 0;
END_IF

IF m_values[i_id].DataType = EDataType.numeric THEN
	m_values[i_id].Value.Numeric := i_value;
	UpdateState_Numeric := TRUE;
ELSE
	UpdateState_Numeric := FALSE;
END_IF
END_METHOD

METHOD UpdateState_NumericIncrement : BOOL
VAR_INPUT
	i_id: UINT;
	
	// writes even if the existing data type does not match
	i_force: BOOL;
END_VAR
IF i_force THEN
	m_values[i_id].DataType := EDataType.numeric;
END_IF

IF m_values[i_id].DataType = EDataType.numeric THEN
	m_values[i_id].Value.Numeric := m_values[i_id].Value.Numeric + 1;
	UpdateState_NumericIncrement := TRUE;
ELSE
	UpdateState_NumericIncrement := FALSE;
END_IF
END_METHOD

METHOD UpdateState_String : BOOL
VAR_INPUT
	i_id: UINT;
	i_value: STRING;
	
	// writes even if the existing data type does not match
	i_force: BOOL;
END_VAR
IF i_force THEN
	m_values[i_id].DataType := EDataType.string_t;
	m_values[i_id].Value.String_t := '';
END_IF

IF m_values[i_id].DataType = EDataType.string_t THEN
	m_values[i_id].Value.String_t := i_value;
	UpdateState_String := TRUE;
ELSE
	UpdateState_String := FALSE;
END_IF
END_METHOD

END_FUNCTION_BLOCK

// ---- Models/ProcessState/ProcessCondition/ComparisonExpression.TcPOU
{attribute 'OPC.UA.DA.StructuredType' := '1'}
FUNCTION_BLOCK ComparisonExpression IMPLEMENTS IExpression
VAR_INPUT
END_VAR
VAR_OUTPUT
END_VAR
VAR
	m_leftId: UINT;				// the ID of the process variable to compare to
	m_sign: EComparisonType;
	m_right: ValueExpression(EDataType.none, FALSE, 0, '', TRUE);
END_VAR

METHOD FB_init : BOOL
VAR_INPUT
	bInitRetains : BOOL; // if TRUE, the retain variables are initialized (warm start / cold start)
	bInCopyCode : BOOL;  // if TRUE, the instance afterwards gets moved into the copy code (online change)
	
	i_leftId: UINT;				// the ID of the process variable to compare to
	i_sign: EComparisonType;
	
	i_dataType: EDataType;
	i_binaryValue: BOOL;
	i_numericValue: LREAL;
	i_stringValue: STRING;
	i_defined: BOOL;
END_VAR
m_leftId := i_leftId;
m_sign := i_sign;
m_right.FB_init(bInitRetains, bInCopyCode,
	i_dataType, i_binaryValue, i_numericValue, i_stringValue, i_defined);
END_METHOD

METHOD IsTrue : BOOL
VAR_INPUT
	i_ptrProcessState: POINTER TO ProcessState;
END_VAR
VAR
	m_val: SValue;
END_VAR
m_val := i_ptrProcessState^.Retrieve(m_leftId, TRUE);

// for each comparison: return FALSE, if the comparison's opposite is TRUE
CASE m_right.o_value.DataType OF
	EDataType.binary:
		CASE m_sign OF
			EComparisonType.equals:
				IF m_val.Value.Binary <> m_right.o_value.Value.Binary THEN
					IsTrue := FALSE;
					RETURN;
				END_IF
			
			EComparisonType.not_equal:
				IF m_val.Value.Binary = m_right.o_value.Value.Binary THEN
					IsTrue := FALSE;
					RETURN;
				END_IF
			
			ELSE // other comparisons not permitted for Bools
				IsTrue := FALSE;
				RETURN;
		END_CASE
		
	EDataType.numeric:
		CASE m_sign OF
			EComparisonType.equals:
				IF m_val.Value.Numeric <> m_right.o_value.Value.Numeric THEN
					IsTrue := FALSE;
					RETURN;
				END_IF
			
			EComparisonType.greater:
				IF m_val.Value.Numeric <= m_right.o_value.Value.Numeric THEN
					IsTrue := FALSE;
					RETURN;
				END_IF
			
			EComparisonType.greater_eq:
				IF m_val.Value.Numeric < m_right.o_value.Value.Numeric THEN
					IsTrue := FALSE;
					RETURN;
				END_IF
			
			EComparisonType.less:
				IF m_val.Value.Numeric >= m_right.o_value.Value.Numeric THEN
					IsTrue := FALSE;
					RETURN;
				END_IF
			
			EComparisonType.less_eq:
				IF m_val.Value.Numeric > m_right.o_value.Value.Numeric THEN
					IsTrue := FALSE;
					RETURN;
				END_IF
			
			EComparisonType.not_equal:
				IF m_val.Value.Numeric = m_right.o_value.Value.Numeric THEN
					IsTrue := FALSE;
					RETURN;
				END_IF
			
			ELSE // unknown comparison
				IsTrue := FALSE;
				RETURN;
		END_CASE
		
	EDataType.string_t:
		CASE m_sign OF
			EComparisonType.equals:
				IF m_val.Value.String_t <> m_right.o_value.Value.String_t THEN
					IsTrue := FALSE;
					RETURN;
				END_IF
			
			EComparisonType.not_equal:
				IF m_val.Value.String_t = m_right.o_value.Value.String_t THEN
					IsTrue := FALSE;
					RETURN;
				END_IF
			
			ELSE // other comparisons not permitted for Strings
				IsTrue := FALSE;
				RETURN;
		END_CASE
	EDataType.dont_care:
		IsTrue := FALSE;
		RETURN;
	EDataType.none:
		IsTrue := FALSE;
		RETURN;
END_CASE

IsTrue := TRUE;
END_METHOD

METHOD ToString : STRING(256)
VAR_INPUT
END_VAR
CASE m_sign OF
	EComparisonType.equals:
		ToString := CONCAT(TO_STRING(m_leftId), CONCAT('#=', m_right.ToString()));
		
	EComparisonType.greater:
		ToString := CONCAT(TO_STRING(m_leftId), CONCAT('#>', m_right.ToString()));
		
	EComparisonType.greater_eq:
		ToString := CONCAT(TO_STRING(m_leftId), CONCAT('#>=', m_right.ToString()));
		
	EComparisonType.less:
		ToString := CONCAT(TO_STRING(m_leftId), CONCAT('#<', m_right.ToString()));
		
	EComparisonType.less_eq:
		ToString := CONCAT(TO_STRING(m_leftId), CONCAT('#<=', m_right.ToString()));
		
	EComparisonType.not_equal:
		ToString := CONCAT(TO_STRING(m_leftId), CONCAT('#<>', m_right.ToString()));
END_CASE
END_METHOD

END_FUNCTION_BLOCK

// ---- Services/Base/ErrorManagerBase.TcPOU
FUNCTION_BLOCK ABSTRACT ErrorManagerBase IMPLEMENTS IService
VAR_INPUT
END_VAR
VAR_OUTPUT
END_VAR
VAR
END_VAR

METHOD ABSTRACT AddMessage : BOOL
VAR_INPUT
	i_alarmId: UINT;
	i_active: BOOL;
	//i_acknowledged: BOOL;
	//i_confirmed: BOOL;
	i_severity: ESeverity;
	//i_retain: BOOL;
	i_instanceName: STRING;
END_VAR
END_METHOD

END_FUNCTION_BLOCK

// ---- Models/Behavior/ModuleSequenceBase.TcPOU
(* Base of Module Sequences. Inheriting FBs must provide the main implementation. *)
FUNCTION_BLOCK ABSTRACT ModuleSequenceBase EXTENDS BehaviorBase
VAR
	m_ptrProcessManager: POINTER TO ProcessManager;
	m_ptrStateTracker: POINTER TO StateTracker;
END_VAR

METHOD ProvideServices : BOOL
VAR_INPUT
	i_ptrProcessManager: POINTER TO ProcessManager;
	i_ptrStateTracker: POINTER TO StateTracker;
END_VAR
THIS^.m_ptrProcessManager := i_ptrProcessManager;
THIS^.m_ptrStateTracker := i_ptrStateTracker;
END_METHOD

METHOD RequestRecovery : BOOL
VAR_INPUT
END_VAR
THIS^.m_ptrProcessManager^.RequestRecovery(THIS^.Postcondition, TO_STRING(m_id));
END_METHOD

END_FUNCTION_BLOCK

// ---- Models/Behavior/LinearSequence.TcPOU
FUNCTION_BLOCK LinearSequence EXTENDS ModuleSequenceBase
VAR_INPUT
	i_primitiveIds: ARRAY [ResiConst.ARR_MIN..ResiConst.MODULE_SEQ_ARR_MAX] OF UINT;
	i_primitiveParams: ARRAY [ResiConst.ARR_MIN..ResiConst.MODULE_SEQ_ARR_MAX] OF ParameterSet;
END_VAR
VAR
	i: UINT;
	
	m_sequenceFinished: BOOL;
	m_primitiveId: UINT;
	m_res: EOperationResult;
END_VAR

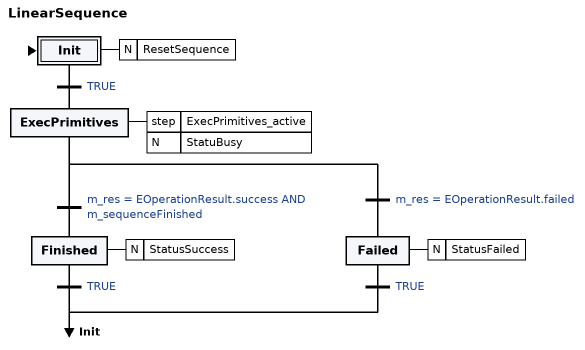
INITIAL_STEP Init:
    ResetSequence(N);
END_STEP
TRANSITION FROM Init TO ExecPrimitives
    := TRUE;
END_TRANSITION
STEP ExecPrimitives:
    ExecPrimitives_active(N);  // step action
    StatuBusy(N);
END_STEP
TRANSITION FROM ExecPrimitives TO Finished
    := m_res = EOperationResult.success AND m_sequenceFinished;
END_TRANSITION
STEP Finished:
    StatusSuccess(N);
END_STEP
TRANSITION FROM Finished TO Init
    := TRUE;
END_TRANSITION
TRANSITION FROM ExecPrimitives TO Failed
    := m_res = EOperationResult.failed;
END_TRANSITION
STEP Failed:
    StatusFailed(N);
END_STEP
TRANSITION FROM Failed TO Init
    := TRUE;
END_TRANSITION

ACTION ExecPrimitives_active:
m_primitiveId := i_primitiveIds[i];

IF m_primitiveId = ESpecialBehaviorIds.empty THEN
	m_sequenceFinished := TRUE;
ELSE
	m_res := m_ptrProcessManager^.Execute(
		i_type := EBehaviorType.control_primitive,
		i_id := m_primitiveId,
		i_params := i_primitiveParams[i]);
		
	IF m_res = EOperationResult.success THEN
		i := i + 1;
	END_IF
END_IF
END_ACTION

PROPERTY Postcondition : IExpression
GET
VAR
	i: UINT;
END_VAR
FOR i := ResiConst.ARR_MIN TO ResiConst.MODULE_SEQ_ARR_MAX DO
	// find the postcondition of the last defined primitive
	IF i_primitiveIds[i] = ESpecialBehaviorIds.empty THEN
		Postcondition := m_ptrProcessManager^.GetBehaviorPtr(EBehaviorType.control_primitive, i_primitiveIds[i - 1])^.Postcondition;
		RETURN;
	END_IF
END_FOR
END_GET
END_PROPERTY

PROPERTY Precondition : IExpression
GET
// precondition of the first defined primitive
Precondition := m_ptrProcessManager^.GetBehaviorPtr(EBehaviorType.control_primitive, i_primitiveIds[ResiConst.ARR_MIN])^.Precondition;
END_GET
END_PROPERTY

METHOD Reset : BOOL
VAR_INPUT
END_VAR
i := ResiConst.ARR_MIN;
m_sequenceFinished := FALSE;
END_METHOD

ACTION ResetSequence:
i := 0;
m_sequenceFinished := FALSE;
m_primitiveId := 0;
o_status := EOperationResult.none;
END_ACTION

ACTION StatuBusy:
o_status := EOperationResult.busy;
END_ACTION

ACTION StatusFailed:
o_status := EOperationResult.failed;
END_ACTION

ACTION StatusSuccess:
o_status := EOperationResult.success;
END_ACTION

END_FUNCTION_BLOCK

// ---- Models/ProcessState/ProcessCondition/BoolExpression.TcPOU
{attribute 'OPC.UA.DA.StructuredType' := '1'}
FUNCTION_BLOCK BoolExpression IMPLEMENTS IExpression
VAR_INPUT
END_VAR
VAR_OUTPUT
END_VAR
VAR
	m_left: IExpression;
	m_sign: EBoolOperation;
	m_right: IExpression;
END_VAR

METHOD FB_init : BOOL
VAR_INPUT
	bInitRetains : BOOL; // if TRUE, the retain variables are initialized (warm start / cold start)
	bInCopyCode : BOOL;  // if TRUE, the instance afterwards gets moved into the copy code (online change)

	i_left: IExpression;
	i_sign: EBoolOperation;
	i_right: IExpression;
END_VAR
m_left := i_left;
m_sign := i_sign;
m_right := i_right;
END_METHOD

METHOD IsTrue : BOOL
VAR_INPUT
	i_ptrProcessState: POINTER TO ProcessState;
END_VAR
CASE m_sign OF
	EBoolOperation.none:
	IsTrue := FALSE;
	
	EBoolOperation.and_op:
	IsTrue := m_left.IsTrue(i_ptrProcessState) AND m_right.IsTrue(i_ptrProcessState);
	
	EBoolOperation.nand_op:
	IsTrue := m_left.IsTrue(i_ptrProcessState) AND NOT m_right.IsTrue(i_ptrProcessState);
	
	EBoolOperation.or_op:
	IsTrue := m_left.IsTrue(i_ptrProcessState) OR m_right.IsTrue(i_ptrProcessState);
		
	EBoolOperation.nor_op:
	IsTrue := m_left.IsTrue(i_ptrProcessState) OR NOT m_right.IsTrue(i_ptrProcessState);
END_CASE
END_METHOD

METHOD ToString : STRING(256)
VAR_INPUT
END_VAR
CASE m_sign OF
	EBoolOperation.and_op:
		ToString := CONCAT('(', CONCAT(m_left.ToString(), CONCAT(')AND(', CONCAT(m_right.ToString(), ')'))));
	
	EBoolOperation.nand_op:
		ToString := CONCAT('(', CONCAT(m_left.ToString(), CONCAT(')NAND(', CONCAT(m_right.ToString(), ')'))));
	
	EBoolOperation.or_op:
		ToString := CONCAT('(', CONCAT(m_left.ToString(), CONCAT(')OR(', CONCAT(m_right.ToString(), ')'))));
	
	EBoolOperation.nor_op:
		ToString := CONCAT('(', CONCAT(m_left.ToString(), CONCAT(')NOR(', CONCAT(m_right.ToString(), ')'))));
	
	ELSE
		ToString := '';
END_CASE
END_METHOD

END_FUNCTION_BLOCK

// ---- Models/ProcessState/HardwareObservationBase.TcPOU
(* Base of Hardware Observations. Ideally, this is the base of every Hardware Control FB. *)
FUNCTION_BLOCK ABSTRACT HardwareObservationBase
VAR
END_VAR

METHOD ABSTRACT ResetDefinition : BOOL
VAR_INPUT
END_VAR
END_METHOD

(* Update an instance of ProcessState with the part of the process that can be observed by this Hardware Interface. *)
METHOD ABSTRACT UpdateProcessObservation : BOOL
VAR_IN_OUT
	io_processState: ProcessState;
END_VAR
END_METHOD

END_FUNCTION_BLOCK

// ---- Models/ProcessState/ProductBase.TcPOU
FUNCTION_BLOCK ProductBase EXTENDS HardwareObservationBase
VAR CONSTANT
	RES_IDX: UINT := 0;
END_VAR
VAR
	// ***** MODIFIED BY RA *****
	raIn_isRemote: BOOL;
	raIn_prodTypeAdr: SAdsSymbol;	// points to the remote's product type (at m_vals[RES_IDX].Values.Numeric)
	raIn_copiedTypeAdr: SAdsSymbol;	// points to the remote's m_copiedProdType
	raIn_resetAdr: SAdsSymbol;		// points to the remote's reset flag
	// **************************
	
	// ***** INIT BY RA OR SUBCLASS *****
	raIn_processStateIdx: UINT;
	// **********************************

	// an array of values characterizing the product. At RES_IDX=0, there is an aggregated "product type"
	m_vals: ARRAY [ResiConst.ARR_MIN..ResiConst.DEFAULT_ARR_MAX] OF SValue;
	// a number (may be an ENUM) defining the type of product. NOTE: 0 means null/nil/None.
	m_copiedProdType: LREAL;
	
	m_valReader: ADSREAD;
	m_copyTrigWriter: ADSWRITE;
	m_resetWriter: ADSWRITE;
	
	// flags
	m_resetPending: BOOL;
	m_defResetPending: BOOL;
	m_trueVal: BOOL := TRUE;
END_VAR

METHOD Copy : BOOL
VAR_INPUT
	i_ptrOther: POINTER TO ProductBase;
END_VAR
Copy := FALSE;

IF NOT raIn_isRemote THEN
	m_copiedProdType := i_ptrOther^.m_vals[RES_IDX].Value.Numeric;
ELSE
	// trigger the remote to do a copy operation
	m_copyTrigWriter(
		NETID := raIn_copiedTypeAdr.NetId,
		PORT := raIn_copiedTypeAdr.Port,
		IDXGRP := raIn_copiedTypeAdr.IdxGrp,
		IDXOFFS := raIn_copiedTypeAdr.IdxOffs,
		LEN := SIZEOF(i_ptrOther^.m_vals[RES_IDX].Value.Numeric),
		SRCADDR := ADR(i_ptrOther^.m_vals[RES_IDX].Value.Numeric),
		WRITE := TRUE);
END_IF

IF NOT m_copyTrigWriter.BUSY THEN
	m_copyTrigWriter(WRITE := FALSE);
	Copy := TRUE;
END_IF
END_METHOD

METHOD Reset : BOOL
m_resetPending := TRUE;
END_METHOD

METHOD ResetConfiguration : BOOL
VAR
	emptySym: SAdsSymbol;
END_VAR
raIn_processStateIdx := 0;

raIn_copiedTypeAdr := emptySym;
raIn_prodTypeAdr := emptySym;
raIn_resetAdr := emptySym;
END_METHOD

METHOD ResetDefinition : BOOL
m_defResetPending := TRUE;
END_METHOD

(* Based on the aggregated product type value, set the separete input values for a consistent shift register. *)
METHOD ReverseSetInputs : BOOL
// not required for the ProductBase
END_METHOD

(* Update an instance of ProcessState with the part of the process that can be observed by this Hardware Interface. *)
METHOD UpdateProcessObservation : BOOL
VAR_IN_OUT
	io_processState: ProcessState;
END_VAR
VAR
	emptyVals: ARRAY [ResiConst.ARR_MIN..ResiConst.DEFAULT_ARR_MAX] OF SValue;
END_VAR
IF raIn_processStateIdx = 0 OR m_copyTrigWriter.BUSY THEN
	RETURN;
END_IF

IF m_copiedProdType <> 0 THEN
	m_vals[RES_IDX].Defined := TRUE;
	m_vals[RES_IDX].DataType := EDataType.numeric;
	m_vals[RES_IDX].Value.Numeric := m_copiedProdType;
	
	ReverseSetInputs();
	m_copiedProdType := 0;
END_IF

// only the aggregated product type (if defined) is copied to the process state, not individual input values
io_processState.SetValue(raIn_processStateIdx, m_vals[RES_IDX]);

// deal with reset requests
m_resetWriter();	// read takes multiple cycles
IF m_resetPending THEN
	IF raIn_isRemote THEN
		// set the remote's reset flag (the local instance will be synced below)
		m_resetWriter(WRITE := FALSE);
		m_resetWriter(
			NETID := raIn_resetAdr.NetId,
			PORT := raIn_resetAdr.Port,
			IDXGRP := raIn_resetAdr.IdxGrp,
			IDXOFFS := raIn_resetAdr.IdxOffs,
			LEN := SIZEOF(m_trueVal),
			SRCADDR := ADR(m_trueVal),
			WRITE := TRUE);
	ELSE
		m_vals[RES_IDX].Value.Numeric := 0;
	END_IF
	
	m_resetPending := FALSE;
	RETURN;
END_IF

// update this product base with the remote's value
IF raIn_isRemote THEN
	// TODO - other data types and potentially multiple result values
	m_vals[RES_IDX].Defined := TRUE;
	m_vals[RES_IDX].DataType := EDataType.numeric;

	m_valReader(READ := FALSE);
	m_valReader(
		NETID := raIn_prodTypeAdr.NetId,
		PORT := raIn_prodTypeAdr.Port,
		IDXGRP := raIn_prodTypeAdr.IdxGrp,
		IDXOFFS := raIn_prodTypeAdr.IdxOffs,
		LEN := SIZEOF(m_vals[RES_IDX].Value.Numeric),
		DESTADDR := ADR(m_vals[RES_IDX].Value.Numeric),
		READ := TRUE);
END_IF
END_METHOD

END_FUNCTION_BLOCK

// ---- Services/ServiceContainer.TcPOU
(*
 * Contains every service relevant to Resi4MPM control.
 * Used so that the services can use each other (similar to dependency injection).
 *)
FUNCTION_BLOCK ServiceContainer
VAR_INPUT
END_VAR
VAR_OUTPUT
END_VAR
VAR
	m_ptrErrorMgr: POINTER TO ErrorManagerBase;
	
	m_pm: ProcessManager;
	m_ptrProcessManager: POINTER TO ProcessManager := ADR(m_pm);
 
	m_st: StateTracker;
	m_ptrStateTracker: POINTER TO StateTracker := ADR(m_st);
END_VAR

METHOD FB_init : BOOL
VAR_INPUT
	bInitRetains : BOOL; // if TRUE, the retain variables are initialized (warm start / cold start)
	bInCopyCode : BOOL;  // if TRUE, the instance afterwards gets moved into the copy code (online change)
	
	i_ptrErrorMgr: POINTER TO ErrorManagerBase;
END_VAR
// get the APPLICATION-SPECIFIC services
THIS^.m_ptrErrorMgr := i_ptrErrorMgr;

// initialize all services
THIS^.m_ptrProcessManager^.ProvideServices(THIS^.m_ptrStateTracker, i_ptrErrorMgr);
THIS^.m_ptrStateTracker^.ProvideServices(THIS^.m_ptrProcessManager);
END_METHOD

PROPERTY PtrErrorManager : POINTER TO ErrorManagerBase
GET
PtrErrorManager := this^.m_ptrErrorMgr;
END_GET
END_PROPERTY

PROPERTY PtrProcessManager : POINTER TO ProcessManager
GET
PtrProcessManager := THIS^.m_ptrProcessManager;
END_GET
END_PROPERTY

PROPERTY PtrStateTracker : POINTER TO StateTracker
GET
PtrStateTracker := THIS^.m_ptrStateTracker;
END_GET
END_PROPERTY

END_FUNCTION_BLOCK
